IF st_config_achse.b_config_fertig THEN
	(* Fehlermeldungen und Betriebsmeldungen ab dem Startindex in die globalen Meldungsarrays schreiben *)
	garr_stoermeldungen[st_config_achse.i16_meld_startindex + 0] := st_sm.b_achse_nicht_bb;
	garr_stoermeldungen[st_config_achse.i16_meld_startindex + 1] := st_sm.b_achse_nicht_referenziert;
	garr_stoermeldungen[st_config_achse.i16_meld_startindex + 2] := st_sm.b_keine_verfahrfreigabe;
	garr_stoermeldungen[st_config_achse.i16_meld_startindex + 3] := st_sm.b_achse_nicht_auf_startpos;
	garr_stoermeldungen[st_config_achse.i16_meld_startindex + 4] := st_sm.b_ende_skalierungs_nocke;
	garr_stoermeldungen[st_config_achse.i16_meld_startindex + 5] := st_sm.b_ende_camming_nocke;
	garr_stoermeldungen[st_config_achse.i16_meld_startindex + 6] := st_sm.b_skalierung_noch_aktiv;
	garr_stoermeldungen[st_config_achse.i16_meld_startindex + 7] := FALSE;
	garr_stoermeldungen[st_config_achse.i16_meld_startindex + 8] := sm_bandrueckzug;
	garr_stoermeldungen[st_config_achse.i16_meld_startindex + 9] := sm_bandreferenzieren;
	garr_stoermeldungen[st_config_achse.i16_meld_startindex + 10] := sm_fehler_bandvorschub;
	garr_stoermeldungen[st_config_achse.i16_meld_startindex + 11] := sm_fehler_raster;
	garr_stoermeldungen[st_config_achse.i16_meld_startindex + 12] := sm_fehler_bandeinfaedeln;
	garr_stoermeldungen[st_config_achse.i16_meld_startindex + 13] := sm_fahren_auf_gls;
	garr_stoermeldungen[st_config_achse.i16_meld_startindex + 14] := sm_band_rausgezogen;
	garr_stoermeldungen[st_config_achse.i16_meld_startindex + 15] := sm_band_nicht_in_lichtschranke;
	garr_stoermeldungen[st_config_achse.i16_meld_startindex + 16] := st_drive_cmd.meldungen.sm_write_soe_parameter;
	garr_stoermeldungen[st_config_achse.i16_meld_startindex + 17] := st_drive_cmd.meldungen.sm_read_soe_parameter;
	garr_stoermeldungen[st_config_achse.i16_meld_startindex + 18] := st_drive_cmd.meldungen.sm_write_nc_parameter;
	garr_stoermeldungen[st_config_achse.i16_meld_startindex + 19] := st_drive_cmd.meldungen.sm_read_nc_parameter;
	garr_stoermeldungen[st_config_achse.i16_meld_startindex + 20] := st_drive_cmd.meldungen.sm_power_enable;
	garr_stoermeldungen[st_config_achse.i16_meld_startindex + 21] := st_drive_cmd.meldungen.sm_power_disable;
	garr_stoermeldungen[st_config_achse.i16_meld_startindex + 22] := st_drive_cmd.meldungen.sm_reset;
	garr_stoermeldungen[st_config_achse.i16_meld_startindex + 23] := st_drive_cmd.meldungen.sm_home;
	garr_stoermeldungen[st_config_achse.i16_meld_startindex + 24] := st_drive_cmd.meldungen.sm_setposition;
	garr_stoermeldungen[st_config_achse.i16_meld_startindex + 25] := st_drive_cmd.meldungen.sm_jog_vorwaerts;
	garr_stoermeldungen[st_config_achse.i16_meld_startindex + 26] := st_drive_cmd.meldungen.sm_jog_rueckwaerts;
	garr_stoermeldungen[st_config_achse.i16_meld_startindex + 27] := st_drive_cmd.meldungen.sm_move_absolute;
	garr_stoermeldungen[st_config_achse.i16_meld_startindex + 28] := st_drive_cmd.meldungen.sm_move_relative;
	garr_stoermeldungen[st_config_achse.i16_meld_startindex + 29] := st_drive_cmd.meldungen.sm_move_velocity;
	garr_stoermeldungen[st_config_achse.i16_meld_startindex + 30] := st_drive_cmd.meldungen.sm_move_modulo;
	garr_stoermeldungen[st_config_achse.i16_meld_startindex + 31] := st_drive_cmd.meldungen.sm_stop_axis;
	garr_stoermeldungen[st_config_achse.i16_meld_startindex + 32] := st_drive_cmd.meldungen.sm_halt_axis;
	garr_stoermeldungen[st_config_achse.i16_meld_startindex + 33] := st_drive_cmd.meldungen.sm_motion_command_timeout;
	garr_stoermeldungen[st_config_achse.i16_meld_startindex + 34] := st_sm.b_achsfehler;
	garr_stoermeldungen[st_config_achse.i16_meld_startindex + 35] := st_sm.b_devicefehler;
	garr_stoermeldungen[st_config_achse.i16_meld_startindex + 36] := st_drive_cmd.meldungen.sm_limit_positiv_erreicht;
	garr_stoermeldungen[st_config_achse.i16_meld_startindex + 37] := st_drive_cmd.meldungen.sm_limit_negativ_erreicht;
	garr_stoermeldungen[st_config_achse.i16_meld_startindex + 38] := st_drive_cmd.meldungen.sm_ec_coe_sdo_write_ex;
	garr_stoermeldungen[st_config_achse.i16_meld_startindex + 39] := st_drive_cmd.meldungen.sm_ec_coe_sdo_read_ex;
	garr_stoermeldungen[st_config_achse.i16_meld_startindex + 40] := FALSE;
	garr_stoermeldungen[st_config_achse.i16_meld_startindex + 41] := FALSE;
	garr_stoermeldungen[st_config_achse.i16_meld_startindex + 42] := FALSE;
	garr_stoermeldungen[st_config_achse.i16_meld_startindex + 43] := FALSE;
	garr_stoermeldungen[st_config_achse.i16_meld_startindex + 44] := FALSE;
	garr_stoermeldungen[st_config_achse.i16_meld_startindex + 45] := FALSE;
	garr_stoermeldungen[st_config_achse.i16_meld_startindex + 46] := FALSE;
	garr_stoermeldungen[st_config_achse.i16_meld_startindex + 47] := FALSE;
	garr_stoermeldungen[st_config_achse.i16_meld_startindex + 49] := FALSE;
	garr_stoermeldungen[st_config_achse.i16_meld_startindex + 50] := FALSE;
	garr_stoermeldungen[st_config_achse.i16_meld_startindex + 51] := FALSE;
	garr_stoermeldungen[st_config_achse.i16_meld_startindex + 52] := FALSE;
	garr_stoermeldungen[st_config_achse.i16_meld_startindex + 53] := FALSE;
	garr_stoermeldungen[st_config_achse.i16_meld_startindex + 54] := FALSE;
	garr_stoermeldungen[st_config_achse.i16_meld_startindex + 55] := FALSE;
	garr_stoermeldungen[st_config_achse.i16_meld_startindex + 56] := FALSE;
	garr_stoermeldungen[st_config_achse.i16_meld_startindex + 57] := FALSE;
	garr_stoermeldungen[st_config_achse.i16_meld_startindex + 58] := FALSE;
	garr_stoermeldungen[st_config_achse.i16_meld_startindex + 59] := FALSE;
	garr_stoermeldungen[st_config_achse.i16_meld_startindex + 60] := FALSE;
	garr_stoermeldungen[st_config_achse.i16_meld_startindex + 61] := FALSE;
	garr_stoermeldungen[st_config_achse.i16_meld_startindex + 62] := FALSE;
	garr_stoermeldungen[st_config_achse.i16_meld_startindex + 63] := FALSE;
	garr_stoermeldungen[st_config_achse.i16_meld_startindex + 64] := FALSE;
	garr_stoermeldungen[st_config_achse.i16_meld_startindex + 65] := FALSE;
	garr_stoermeldungen[st_config_achse.i16_meld_startindex + 66] := FALSE;
	garr_stoermeldungen[st_config_achse.i16_meld_startindex + 67] := FALSE;
	garr_stoermeldungen[st_config_achse.i16_meld_startindex + 68] := FALSE;
	garr_stoermeldungen[st_config_achse.i16_meld_startindex + 69] := FALSE;
	garr_stoermeldungen[st_config_achse.i16_meld_startindex + 70] := FALSE;
	garr_stoermeldungen[st_config_achse.i16_meld_startindex + 71] := FALSE;
	garr_stoermeldungen[st_config_achse.i16_meld_startindex + 72] := FALSE;
	garr_stoermeldungen[st_config_achse.i16_meld_startindex + 73] := FALSE;
	garr_stoermeldungen[st_config_achse.i16_meld_startindex + 74] := FALSE;
	garr_stoermeldungen[st_config_achse.i16_meld_startindex + 75] := FALSE;
	garr_stoermeldungen[st_config_achse.i16_meld_startindex + 76] := FALSE;
	garr_stoermeldungen[st_config_achse.i16_meld_startindex + 77] := FALSE;
	garr_stoermeldungen[st_config_achse.i16_meld_startindex + 78] := FALSE;
	garr_stoermeldungen[st_config_achse.i16_meld_startindex + 79] := FALSE;
	garr_stoermeldungen[st_config_achse.i16_meld_startindex + 80] := FALSE;
	garr_stoermeldungen[st_config_achse.i16_meld_startindex + 81] := FALSE;
	garr_stoermeldungen[st_config_achse.i16_meld_startindex + 82] := FALSE;
	garr_stoermeldungen[st_config_achse.i16_meld_startindex + 83] := FALSE;
	garr_stoermeldungen[st_config_achse.i16_meld_startindex + 84] := FALSE;
	garr_stoermeldungen[st_config_achse.i16_meld_startindex + 85] := FALSE;
	garr_stoermeldungen[st_config_achse.i16_meld_startindex + 86] := FALSE;
	garr_stoermeldungen[st_config_achse.i16_meld_startindex + 87] := FALSE;
	garr_stoermeldungen[st_config_achse.i16_meld_startindex + 88] := FALSE;
	garr_stoermeldungen[st_config_achse.i16_meld_startindex + 89] := FALSE;
	garr_stoermeldungen[st_config_achse.i16_meld_startindex + 90] := FALSE;
	garr_stoermeldungen[st_config_achse.i16_meld_startindex + 91] := FALSE;
	garr_stoermeldungen[st_config_achse.i16_meld_startindex + 92] := FALSE;
	garr_stoermeldungen[st_config_achse.i16_meld_startindex + 93] := FALSE;
	garr_stoermeldungen[st_config_achse.i16_meld_startindex + 94] := FALSE;
	garr_stoermeldungen[st_config_achse.i16_meld_startindex + 95] := FALSE;
	garr_stoermeldungen[st_config_achse.i16_meld_startindex + 96] := FALSE;
	garr_stoermeldungen[st_config_achse.i16_meld_startindex + 97] := FALSE;
	garr_stoermeldungen[st_config_achse.i16_meld_startindex + 98] := FALSE;
	garr_stoermeldungen[st_config_achse.i16_meld_startindex + 99] := FALSE;
	
	garr_betriebsmeldungen[st_config_achse.i16_meld_startindex + 0] := FALSE;
	garr_betriebsmeldungen[st_config_achse.i16_meld_startindex + 1] := FALSE;
	garr_betriebsmeldungen[st_config_achse.i16_meld_startindex + 2] := FALSE;
	garr_betriebsmeldungen[st_config_achse.i16_meld_startindex + 3] := FALSE;
	garr_betriebsmeldungen[st_config_achse.i16_meld_startindex + 4] := FALSE;
	garr_betriebsmeldungen[st_config_achse.i16_meld_startindex + 5] := FALSE;
	garr_betriebsmeldungen[st_config_achse.i16_meld_startindex + 6] := FALSE;
	garr_betriebsmeldungen[st_config_achse.i16_meld_startindex + 7] := FALSE;
	garr_betriebsmeldungen[st_config_achse.i16_meld_startindex + 8] := FALSE;
	garr_betriebsmeldungen[st_config_achse.i16_meld_startindex + 9] := FALSE;
	garr_betriebsmeldungen[st_config_achse.i16_meld_startindex + 10] := FALSE;
	garr_betriebsmeldungen[st_config_achse.i16_meld_startindex + 11] := FALSE;
	garr_betriebsmeldungen[st_config_achse.i16_meld_startindex + 12] := FALSE;
	garr_betriebsmeldungen[st_config_achse.i16_meld_startindex + 13] := FALSE;
	garr_betriebsmeldungen[st_config_achse.i16_meld_startindex + 14] := FALSE;
	garr_betriebsmeldungen[st_config_achse.i16_meld_startindex + 15] := FALSE;
	garr_betriebsmeldungen[st_config_achse.i16_meld_startindex + 16] := FALSE;
	garr_betriebsmeldungen[st_config_achse.i16_meld_startindex + 17] := FALSE;
	garr_betriebsmeldungen[st_config_achse.i16_meld_startindex + 18] := FALSE;
	garr_betriebsmeldungen[st_config_achse.i16_meld_startindex + 19] := FALSE;
	garr_betriebsmeldungen[st_config_achse.i16_meld_startindex + 20] := FALSE;
	garr_betriebsmeldungen[st_config_achse.i16_meld_startindex + 21] := FALSE;
	garr_betriebsmeldungen[st_config_achse.i16_meld_startindex + 22] := FALSE;
	garr_betriebsmeldungen[st_config_achse.i16_meld_startindex + 23] := FALSE;
	garr_betriebsmeldungen[st_config_achse.i16_meld_startindex + 24] := FALSE;
	garr_betriebsmeldungen[st_config_achse.i16_meld_startindex + 25] := FALSE;
	garr_betriebsmeldungen[st_config_achse.i16_meld_startindex + 26] := FALSE;
	garr_betriebsmeldungen[st_config_achse.i16_meld_startindex + 27] := FALSE;
	garr_betriebsmeldungen[st_config_achse.i16_meld_startindex + 28] := FALSE;
	garr_betriebsmeldungen[st_config_achse.i16_meld_startindex + 29] := FALSE;
	garr_betriebsmeldungen[st_config_achse.i16_meld_startindex + 30] := FALSE;
	garr_betriebsmeldungen[st_config_achse.i16_meld_startindex + 31] := FALSE;
	garr_betriebsmeldungen[st_config_achse.i16_meld_startindex + 32] := FALSE;
	garr_betriebsmeldungen[st_config_achse.i16_meld_startindex + 33] := FALSE;
	garr_betriebsmeldungen[st_config_achse.i16_meld_startindex + 34] := FALSE;
	garr_betriebsmeldungen[st_config_achse.i16_meld_startindex + 35] := FALSE;
	garr_betriebsmeldungen[st_config_achse.i16_meld_startindex + 36] := FALSE;
	garr_betriebsmeldungen[st_config_achse.i16_meld_startindex + 37] := FALSE;
	garr_betriebsmeldungen[st_config_achse.i16_meld_startindex + 38] := FALSE;
	garr_betriebsmeldungen[st_config_achse.i16_meld_startindex + 39] := FALSE;
	garr_betriebsmeldungen[st_config_achse.i16_meld_startindex + 40] := FALSE;
	garr_betriebsmeldungen[st_config_achse.i16_meld_startindex + 41] := FALSE;
	garr_betriebsmeldungen[st_config_achse.i16_meld_startindex + 42] := FALSE;
	garr_betriebsmeldungen[st_config_achse.i16_meld_startindex + 43] := FALSE;
	garr_betriebsmeldungen[st_config_achse.i16_meld_startindex + 44] := FALSE;
	garr_betriebsmeldungen[st_config_achse.i16_meld_startindex + 45] := FALSE;
	garr_betriebsmeldungen[st_config_achse.i16_meld_startindex + 46] := FALSE;
	garr_betriebsmeldungen[st_config_achse.i16_meld_startindex + 47] := FALSE;
	garr_betriebsmeldungen[st_config_achse.i16_meld_startindex + 48] := FALSE;
	garr_betriebsmeldungen[st_config_achse.i16_meld_startindex + 49] := FALSE;
END_IF
END_PROGRAM
ACTION subr_ST_Vorschubkontrolle:
IF gi16_betriebsart <> HAND AND NOT ST_TippTasten.b_einfaedeln_aktiv AND st_ctrl_in.b_freigabe THEN
(* Warte auf Vorschubnocke  und Freigabe von der Virtuellen Masterachse *)
(* Die Freigabe erfolgt nur im normalen Produktionsablauf; nicht bei Bandwechsel, Einfädeln, ... da hier keine Überwachung erfolgen soll. *)

	(* Am Anfang des Bandvorschubs Zähler zurücksetzen *)
	IF  fb_r_trig_nocke_einzug.Q THEN
		i_zaehler_steigende_flanke := 0;
		i_zaehler_fallende_flanke := 0;
	END_IF

	(* Zähler Vorschubkontrolle durch positive Flanke erhöhen *)
	IF fb_r_trig_vorschubkontrolle.Q THEN
		i_zaehler_steigende_flanke := i_zaehler_steigende_flanke + 1;
	END_IF
	(* Zähler Vorschubkontrolle durch negative Flanke erhöhen *)
	IF fb_f_trig_vorschubkontrolle.Q THEN
		i_zaehler_fallende_flanke := i_zaehler_fallende_flanke + 1;
	END_IF

	(* Am Ende des Bandvorschubs die Zähler mit der Vorgabe vergleichen *)
	IF fb_f_trig_nocke_einzug.Q THEN
		IF 	i_zaehler_steigende_flanke <> gst_datensatz.st_bestueckprogramm.i16_b[ST_Virtuelle_Masterachse.i16_bestueckposzaehler] OR
			i_zaehler_fallende_flanke <> gst_datensatz.st_bestueckprogramm.i16_b[ST_Virtuelle_Masterachse.i16_bestueckposzaehler] THEN
			sm_fehler_bandvorschub := TRUE;
			fb_state_entry.i16_next_step := FEHLER;
		END_IF
	END_IF
ELSE
	i_zaehler_steigende_flanke := 0;
	i_zaehler_fallende_flanke := 0;
END_IF
END_ACTION

(* POU Gemeinsamkeiten17xx/Betriebsarten/ST_Betriebsarten, ST *)
PROGRAM ST_Betriebsarten
VAR_INPUT
	st_config					: struct_config;
END_VAR
VAR
	fb_ton_wz				: TON;
	fb_state_entry				: ST_StateEntry;
	i16_betriebsart 			: enum_betriebsarten := KEINE;
	e_ba_automatik			AT %I* : BOOL;
	e_ba_tippen				AT %I* : BOOL;
	e_ba_hand				AT %I* : BOOL;
	e_ba_dummy				AT %I* : BOOL;
	e_ba_pseudo			AT %I* : BOOL;
	a_lampe_ba_automatik	AT %Q* : BOOL;
	a_lampe_ba_tippen		AT %Q* : BOOL;
	a_lampe_ba_hand		AT %Q* : BOOL;
	a_lampe_ba_dummy		AT %Q* : BOOL;
	a_lampe_ba_pseudo		AT %Q* : BOOL;
END_VAR
gi16_betriebsart := i16_betriebsart;

(* Zeiten *)
fb_ton_wz(IN:= , PT:= t#1s, Q=>  , ET=> );

(* ======================================Schrittkette======================================== *)
fb_state_entry(
	i16_next_step:= ,
	i16_pos:= 1,
	s_debugtext:= ,
	E=> ,
	X=> ,
	i16_step=> ,
	i16_last_step=> );

CASE fb_state_entry.i16_step OF
(*=======================================================*)
	0:	(* KEINE *)
		IF fb_state_entry.E THEN
			fb_ton_wz.IN := TRUE;
		END_IF
		IF fb_ton_wz.Q THEN
			i16_betriebsart := KEINE;
		END_IF

		a_lampe_ba_automatik := FALSE;
		a_lampe_ba_tippen := FALSE;
		a_lampe_ba_hand := FALSE;
		a_lampe_ba_dummy := FALSE;
		a_lampe_ba_pseudo := FALSE;

		(* Betriebsartenwechsel *)
		IF e_ba_automatik THEN
			fb_state_entry.i16_next_step := 10;	(* AUTO *)
		ELSIF e_ba_tippen THEN
			fb_state_entry.i16_next_step := 20;	(* TIPPEN *)
		ELSIF e_ba_hand THEN
			fb_state_entry.i16_next_step := 30;	(* HAND *)
		ELSIF e_ba_dummy THEN
			fb_state_entry.i16_next_step := 40;	(* DUMMY *)
		ELSIF e_ba_pseudo THEN
			fb_state_entry.i16_next_step := 50;	(* PSEUDO *)
		END_IF

(*=======================================================*)
	10:	(* AUTO *)
		IF fb_state_entry.E THEN
			i16_betriebsart := AUTO;
			a_lampe_ba_automatik := TRUE;
		END_IF

		(* Betriebsartenwechsel *)
		IF NOT e_ba_automatik THEN
			fb_state_entry.i16_next_step := 0;
		END_IF
	
	(*=======================================================*)
	20:	(* TIPPEN *)
		IF fb_state_entry.E THEN
			i16_betriebsart := TIPPEN;
			a_lampe_ba_tippen := TRUE;
		END_IF

		(* Betriebsartenwechsel *)
		IF NOT e_ba_tippen THEN
			fb_state_entry.i16_next_step := 0;
		END_IF

(*=======================================================*)
	30:	(* HAND *)
		IF fb_state_entry.E THEN
			i16_betriebsart := HAND;
			a_lampe_ba_hand := TRUE;
		END_IF

		(* Betriebsartenwechsel *)
		IF NOT e_ba_hand THEN
			fb_state_entry.i16_next_step := 0;
		END_IF

(*=======================================================*)
	40:	(* DUMMY *)
		IF fb_state_entry.E THEN
			i16_betriebsart := DUMMY;
			a_lampe_ba_dummy := TRUE;
		END_IF

		(* Betriebsartenwechsel *)
		IF NOT e_ba_dummy THEN
			fb_state_entry.i16_next_step := 0;
		END_IF

(*=======================================================*)
	50:	(* PSEUDO *)
		IF fb_state_entry.E THEN
			i16_betriebsart := PSEUDO;
			a_lampe_ba_pseudo := TRUE;
		END_IF

		(* Betriebsartenwechsel *)
		IF NOT e_ba_pseudo THEN
			fb_state_entry.i16_next_step := 0;
		END_IF
END_CASE

fb_state_entry(
	i16_next_step:= ,
	i16_pos:= 2,
	s_debugtext:= ,
	E=> , 
	X=> , 
	i16_step=> ,
	i16_last_step=> );

IF st_config.b_config_fertig THEN
	(* Fehlermeldungen  *)
	garr_stoermeldungen[st_config.i16_meld_startindex + 0] := FALSE;
	garr_stoermeldungen[st_config.i16_meld_startindex + 1] := FALSE;
	garr_stoermeldungen[st_config.i16_meld_startindex + 2] := FALSE;
	garr_stoermeldungen[st_config.i16_meld_startindex + 3] := FALSE;
	garr_stoermeldungen[st_config.i16_meld_startindex + 4] := FALSE;
	garr_stoermeldungen[st_config.i16_meld_startindex + 5] := FALSE;
	garr_stoermeldungen[st_config.i16_meld_startindex + 6] := FALSE;
	garr_stoermeldungen[st_config.i16_meld_startindex + 7] := FALSE;
	garr_stoermeldungen[st_config.i16_meld_startindex + 8] := FALSE;
	garr_stoermeldungen[st_config.i16_meld_startindex + 9] := FALSE;
	garr_stoermeldungen[st_config.i16_meld_startindex + 10] := FALSE;
	garr_stoermeldungen[st_config.i16_meld_startindex + 11] := FALSE;
	garr_stoermeldungen[st_config.i16_meld_startindex + 12] := FALSE;
	garr_stoermeldungen[st_config.i16_meld_startindex + 13] := FALSE;
	garr_stoermeldungen[st_config.i16_meld_startindex + 14] := FALSE;
	garr_stoermeldungen[st_config.i16_meld_startindex + 15] := FALSE;
	garr_stoermeldungen[st_config.i16_meld_startindex + 16] := FALSE;
	garr_stoermeldungen[st_config.i16_meld_startindex + 17] := FALSE;
	garr_stoermeldungen[st_config.i16_meld_startindex + 18] := FALSE;
	garr_stoermeldungen[st_config.i16_meld_startindex + 19] := FALSE;
	
	(* Betriebsmeldungen *)
	garr_betriebsmeldungen[st_config.i16_meld_startindex + 0] := FALSE;
	garr_betriebsmeldungen[st_config.i16_meld_startindex + 1] := FALSE;
	garr_betriebsmeldungen[st_config.i16_meld_startindex + 2] := FALSE;
	garr_betriebsmeldungen[st_config.i16_meld_startindex + 3] := FALSE;
	garr_betriebsmeldungen[st_config.i16_meld_startindex + 4] := FALSE;
	garr_betriebsmeldungen[st_config.i16_meld_startindex + 5] := FALSE;
	garr_betriebsmeldungen[st_config.i16_meld_startindex + 6] := FALSE;
	garr_betriebsmeldungen[st_config.i16_meld_startindex + 7] := FALSE;
	garr_betriebsmeldungen[st_config.i16_meld_startindex + 8] := FALSE;
	garr_betriebsmeldungen[st_config.i16_meld_startindex + 9] := FALSE;
	garr_betriebsmeldungen[st_config.i16_meld_startindex + 10] := FALSE;
	garr_betriebsmeldungen[st_config.i16_meld_startindex + 11] := FALSE;
	garr_betriebsmeldungen[st_config.i16_meld_startindex + 12] := FALSE;
	garr_betriebsmeldungen[st_config.i16_meld_startindex + 13] := FALSE;
	garr_betriebsmeldungen[st_config.i16_meld_startindex + 14] := FALSE;
	garr_betriebsmeldungen[st_config.i16_meld_startindex + 15] := FALSE;
	garr_betriebsmeldungen[st_config.i16_meld_startindex + 16] := FALSE;
	garr_betriebsmeldungen[st_config.i16_meld_startindex + 17] := FALSE;
	garr_betriebsmeldungen[st_config.i16_meld_startindex + 18] := FALSE;
	garr_betriebsmeldungen[st_config.i16_meld_startindex + 19] := FALSE;
END_IF
END_PROGRAM

(* POU Gemeinsamkeiten17xx/Achsen/F_Servobandeinzug_Strecke_zu_Grad, ST *)
FUNCTION F_Servobandeinzug_Strecke_zu_Grad : LREAL
VAR_INPUT
	strecke	: LREAL;
END_VAR
VAR
	Umfang : LREAL;
END_VAR
Umfang :=  gst_datensatz.st_band.i16_igelrad_zaehne * gst_datensatz.st_band.r_raster;
lr_debug :=  (360.0 * strecke ) / Umfang ;
F_Servobandeinzug_Strecke_zu_Grad := lr_debug;
END_FUNCTION

(* POU Gemeinsamkeiten17xx/Achsen/F_Startpos_Servobandeinzug, ST *)
FUNCTION F_Startpos_Servobandeinzug : LREAL
VAR_INPUT
	r_actual_pos : LREAL:= 1.0;
END_VAR
VAR
	i16_gerundet : INT:= 0;
	startpos : INT := 3;
	i16_grad_pro_zahn : INT := 10;
	r_grad_pro_zahn : LREAL := 10.0;
END_VAR
(* Das Igelrad muss zum Einfädeln an einer bestimmten Gradzahl stehen.
Diese ist abhängig von der größe des Igelrads *)

i16_gerundet := LREAL_TO_INT(r_actual_pos/r_grad_pro_zahn);

F_Startpos_Servobandeinzug := INT_TO_LREAL(i16_gerundet * i16_grad_pro_zahn - gst_datensatz.st_band.i16_startpos_einfaedeln);
END_FUNCTION

(* POU Gemeinsamkeiten17xx/TagReader/ST_Konvertiere_gelese_TagData, ST *)
PROGRAM ST_Konvertiere_gelese_TagData
VAR
	i : INT := 0;
END_VAR
IF gst_datensatz.st_md.i16_tag_data_structur_version = 0 THEN
	gst_tag_data.WpcNumber := balluff_tag_reader.fb.s_lese_daten[0];
	gst_tag_data.StateParts[0] := balluff_tag_reader.fb.s_lese_daten[1];
	gst_tag_data.StateParts[1] := balluff_tag_reader.fb.s_lese_daten[2];

	MEMCPY( ADR(gst_tag_data.Articelnumber), ADR(balluff_tag_reader.fb.s_lese_daten[3]), 50);
	gst_tag_data.LastUsedTool := balluff_tag_reader.fb.s_lese_daten[54];
	MEMCPY( ADR(gst_tag_data.UmlNo_VPE), ADR(balluff_tag_reader.fb.s_lese_daten[55]), 4);
	gst_datensatz.st_md.s_aktuelle_artikelnummer := gst_tag_data.Articelnumber;
ELSIF gst_datensatz.st_md.i16_tag_data_structur_version = 1 THEN
	gst_tag_data.WpcNumber := balluff_tag_reader.fb.s_lese_daten[0];
	FOR i:= 0 TO 7 BY 1 DO
		gst_tag_data.StateParts[i] := balluff_tag_reader.fb.s_lese_daten[i + 1];
	END_FOR
	gst_tag_data.AmountPartsOnWpc := balluff_tag_reader.fb.s_lese_daten[10];
	gst_tag_data.LastUsedTool := balluff_tag_reader.fb.s_lese_daten[15];
	MEMCPY( ADR(gst_tag_data.Articelnumber), ADR(balluff_tag_reader.fb.s_lese_daten[20]), 50);
	MEMCPY( ADR(gst_tag_data.UmlNo_VPE), ADR(balluff_tag_reader.fb.s_lese_daten[71]), 4);
	gst_datensatz.st_md.s_aktuelle_artikelnummer := gst_tag_data.Articelnumber;
END_IF

(* Wenn Haken in Visu gesetzt ist dann BESTUECKUNG_MANUAL *)
(* Sonst kommt Info von der WT-XML *)
IF gst_datensatz.st_md.b_bestueckprogramm_manuell THEN
	gst_datensatz.st_md.i16_typ_bestueckmodus := BESTUECKUNG_MANUAL;
ELSE
	gst_datensatz.st_md.i16_typ_bestueckmodus := gst_datensatz.st_wt.i16_typ_bestueckmodus;
END_IF

(* Wenn Hublift links aktiv ist, soll Zelle Last Used Tool auf 0 zurücksetzen *)
(* Damit wird UML simuliert. Diese Funktion ermöglicht Kleinserien mit Hublift links *)
IF gst_datensatz.st_md.b_hublift_links_aktiv THEN
	gst_tag_data.StateParts[0] := PART_NEW;
	gst_tag_data.StateParts[1] := PART_NEW;
	gst_tag_data.LastUsedTool := 0;
END_IF
END_PROGRAM

(* POU Gemeinsamkeiten17xx/TagReader/ST_Markiere_WT_NIO, ST *)
PROGRAM ST_Markiere_WT_NIO
VAR
	i : INT := 0;
END_VAR
IF gst_datensatz.st_md.i16_tag_data_structur_version = 0 THEN
	gst_tag_data.StateParts[0] := PART_NOK;
	gst_tag_data.StateParts[1] := PART_NOK;

	(* Starte Schreib Prozess *)
	balluff_tag_reader.fb.i16_addresse := 1;
	balluff_tag_reader.fb.i16_anzahl_byte := 2;
	balluff_tag_reader.fb.s_schreib_daten[0] := DINT_TO_BYTE(gst_tag_data.StateParts[0]);
	balluff_tag_reader.fb.s_schreib_daten[1] := DINT_TO_BYTE(gst_tag_data.StateParts[1]);
	balluff_tag_reader.st_ctrl.in.b_start_schreiben := TRUE;
ELSIF gst_datensatz.st_md.i16_tag_data_structur_version = 1 THEN
	balluff_tag_reader.fb.i16_addresse := 1;
	balluff_tag_reader.fb.i16_anzahl_byte := 8;
	FOR i:= 0 TO gst_tag_data.AmountPartsOnWpc - 1 BY 1 DO
		gst_tag_data.StateParts[i] := PART_NOK;
	END_FOR
	FOR i:= gst_tag_data.AmountPartsOnWpc TO 7 BY 1 DO
		gst_tag_data.StateParts[i] := PART_NO;
	END_FOR
	FOR i:= 0 TO 7 BY 1 DO
		balluff_tag_reader.fb.s_schreib_daten[i] := DINT_TO_BYTE(gst_tag_data.StateParts[i]);
	END_FOR
	balluff_tag_reader.st_ctrl.in.b_start_schreiben := TRUE;
END_IF
END_PROGRAM

(* POU Gemeinsamkeiten17xx/TagReader/ST_Markiere_WT_IO, ST *)
PROGRAM ST_Markiere_WT_IO
VAR
	i 						:INT := 0;
	b_Rasterfolie_montiert	:BOOL;
END_VAR
(* Auswertung der Bestückung (Pins bzw. Rasterplatte) des ISK *)
CASE gst_datensatz.st_md.i16_typ_zelle OF
	KEINE_ZELLE:
		;

	BESTUECKZELLE_1700:
		(* WT Hat die Maschine auf regulärem Weg wieder verlassen *)
		(* --> Teil ist Ok *)
		IF gst_datensatz.st_md.i16_tag_data_structur_version = 0 THEN
			gst_tag_data.StateParts[0] := PART_OK;
			gst_tag_data.StateParts[1] := PART_OK;	(* Damit die Stuktur nicht umgestellt werden muss, bei 2 ISO auf einem WT *)
		ELSIF gst_datensatz.st_md.i16_tag_data_structur_version = 1 THEN
			FOR i:= 0 TO gst_tag_data.AmountPartsOnWpc - 1 BY 1 DO
				gst_tag_data.StateParts[i] := PART_OK;
			END_FOR
			FOR i:= gst_tag_data.AmountPartsOnWpc TO 7 BY 1 DO
				gst_tag_data.StateParts[i] := PART_NO;
			END_FOR
		END_IF

	BESTUECKZELLE_1720:
		(* WT Hat die Maschine auf regulärem Weg wieder verlassen *)
		(* --> Teil ist Ok *)
		IF gst_datensatz.st_md.i16_tag_data_structur_version = 0 THEN
			gst_tag_data.StateParts[0] := PART_OK;
			gst_tag_data.StateParts[1] := PART_OK;
		ELSIF gst_datensatz.st_md.i16_tag_data_structur_version = 1 THEN
			FOR i:= 0 TO gst_tag_data.AmountPartsOnWpc - 1 BY 1 DO
				gst_tag_data.StateParts[i] := PART_OK;
			END_FOR
			FOR i:= gst_tag_data.AmountPartsOnWpc TO 7 BY 1 DO
				gst_tag_data.StateParts[i] := PART_NO;
			END_FOR
		END_IF

	RASTERFOLIE:
			b_Rasterfolie_montiert:=	TRUE;
			FOR i := 0 TO DINT_TO_INT(gst_datensatz.st_bestueckprogramm.i32_anzahl) - 1 BY 1 DO
				IF	NOT ST_Rasterfolienmontage.arr_rafo_schieberegister[i]THEN
					b_Rasterfolie_montiert:=	FALSE;
				END_IF
			END_FOR

		IF gst_datensatz.st_md.i16_tag_data_structur_version = 0 THEN
			IF b_Rasterfolie_montiert THEN
				gst_tag_data.StateParts[0] := PART_OK;
				gst_tag_data.StateParts[1] := PART_OK;	(* Damit die Stuktur nicht umgestellt werden muss, bei 2 ISO auf einem WT *)
			ELSE
				gst_tag_data.StateParts[0] := PART_NOK;
				gst_tag_data.StateParts[1] := PART_NOK;
			END_IF
		ELSIF gst_datensatz.st_md.i16_tag_data_structur_version = 1 THEN
			IF b_Rasterfolie_montiert THEN
				FOR i:= 0 TO gst_tag_data.AmountPartsOnWpc - 1 BY 1 DO
					gst_tag_data.StateParts[i] := PART_OK;
				END_FOR
				FOR i:= gst_tag_data.AmountPartsOnWpc TO 7 BY 1 DO
					gst_tag_data.StateParts[i] := PART_NO;
				END_FOR
			ELSE
				FOR i:= 0 TO gst_tag_data.AmountPartsOnWpc - 1 BY 1 DO
					gst_tag_data.StateParts[i] := PART_NOK;
				END_FOR
				FOR i:= gst_tag_data.AmountPartsOnWpc TO 7 BY 1 DO
					gst_tag_data.StateParts[i] := PART_NO;
				END_FOR
			END_IF
		END_IF
END_CASE
(* Starte Schreib Prozess *)
IF gst_datensatz.st_md.i16_tag_data_structur_version = 0 THEN
	balluff_tag_reader.fb.i16_addresse := 1;
	balluff_tag_reader.fb.i16_anzahl_byte := 2;
	balluff_tag_reader.fb.s_schreib_daten[0] := DINT_TO_BYTE(gst_tag_data.StateParts[0]);
	balluff_tag_reader.fb.s_schreib_daten[1] := DINT_TO_BYTE(gst_tag_data.StateParts[1]);
	balluff_tag_reader.st_ctrl.in.b_start_schreiben := TRUE;
ELSIF gst_datensatz.st_md.i16_tag_data_structur_version = 1THEN
	balluff_tag_reader.fb.i16_addresse := 1;
	balluff_tag_reader.fb.i16_anzahl_byte := 8;
	FOR i:= 0 TO 7 BY 1 DO
		balluff_tag_reader.fb.s_schreib_daten[i] := DINT_TO_BYTE(gst_tag_data.StateParts[i]);
	END_FOR
	balluff_tag_reader.st_ctrl.in.b_start_schreiben := TRUE;
END_IF
END_PROGRAM

(* POU Gemeinsamkeiten17xx/TagReader/ST_Schreibe_LastUsedTool, ST *)
PROGRAM ST_Schreibe_LastUsedTool
VAR
END_VAR
(* Starte Schreib Prozess *)
IF gst_datensatz.st_md.i16_tag_data_structur_version = 0 THEN
	balluff_tag_reader.fb.i16_addresse := 54;
	balluff_tag_reader.fb.i16_anzahl_byte := 1;
	balluff_tag_reader.fb.s_schreib_daten[0] := gst_tag_data.LastUsedTool;
	balluff_tag_reader.st_ctrl.in.b_start_schreiben := TRUE;
ELSIF gst_datensatz.st_md.i16_tag_data_structur_version = 1 THEN
	balluff_tag_reader.fb.i16_addresse := 15;
	balluff_tag_reader.fb.i16_anzahl_byte := 1;
	balluff_tag_reader.fb.s_schreib_daten[0] := gst_tag_data.LastUsedTool;
	balluff_tag_reader.st_ctrl.in.b_start_schreiben := TRUE;
END_IF
END_PROGRAM

(* POU Gemeinsamkeiten17xx/Achsen/ST_Bestueckachse, ST *)
PROGRAM ST_Bestueckachse
VAR_INPUT
	st_config_achse						: struct_ecd_config;
	st_ctrl_in								: struct_ctrl_in;
	e_steuerung_ein						: BOOL;
	e_ba_mit_bedingungen				: BOOL;
	e_tuere_vorne_offen					: BOOL;
	e_tuere_hinten_offen					: BOOL;
END_VAR
VAR_IN_OUT
	st_visu								: struct_ecd_visu;
END_VAR
VAR_OUTPUT
	st_ctrl_out							: struct_ctrl_out;
END_VAR
VAR
	st_sm						 		: struct_ecd_meldungen;
	st_drive_cmd							: struct_ecd_cmd;
	fb_ton_wz							: TON;
	fb_ton_quitt							: TON;
	fb_ton_wz_disable						: TON;
	fb_r_trig_tippen						: R_TRIG;
	fb_f_trig_tippen						: F_TRIG;
	fb_r_trig_taste_plus					: R_TRIG;
	fb_r_trig_taste_minus					: R_TRIG;
	fb_r_trig_start							: R_TRIG;
	fb_r_trig_hand_dialog					: R_TRIG;
	fb_r_trig_nullpunkt_setzen				: R_TRIG;
	fb_axis								: ST_AxisJobCtrl_Motion;
	fb_state_entry							: ST_StateEntry;
	fb_ton_uez							: TON;
	i, j									: INT := 0;
	lr_pos_ohneverschiebung			: LREAL;
	st_geschwindigkeiten					: struct_ecd_geschwindigkeiten;
	b_hand_dialog_aktiv					: BOOL := FALSE;
	b_nullnockenmerker					: BOOL := FALSE;

	sm_fehler_initialposition_achse			: BOOL := FALSE;
	sm_keine_nocken_definiert				: BOOL := FALSE;
	sm_fehler_ot_ut						: BOOL := FALSE;

	e_referenz_sensor						AT %I* : BOOL;
	i16_torque							AT %I* : INT;

	fb_ot_ut_ueberwachung				: ST_OT_UT_Ueberwachung;

	lr_decceleration_nothalt				: LREAL;
	lr_decceleration_normal				: LREAL;
END_VAR
(* Zeiten *)
fb_ton_wz(IN:= ,PT:= , Q=>  , ET=> );
fb_ton_uez(IN:= ,	PT:= , Q=>  , ET=> );
fb_ton_quitt(IN:= , PT:= t#100ms, Q=> , ET=> );
fb_ton_wz_disable(IN:= , PT:= t#500ms, Q=> , ET=> );

(* Flanken *)
fb_r_trig_taste_plus(CLK:= ST_Euchner_Handbedienpult.b_Taste_Plus, Q=> );
fb_r_trig_taste_minus(CLK:= ST_Euchner_Handbedienpult.b_Taste_Minus, Q=> );
fb_r_trig_start(CLK:= st_ctrl_in.b_start, Q=> );
fb_r_trig_hand_dialog(CLK:= b_hand_dialog_aktiv, Q=> );
fb_r_trig_nullpunkt_setzen(CLK:= axis_bestueckachse.st_visu.b_nullpunkt_setzen, Q=> );

(* Achse steuern *)
(* Bestueckachse *)
fb_axis(
	e_referenznocken:= ,
	b_refsensor_vorhanden:= st_config_achse.b_refsensor_vorhanden,
	b_limitsensor_positiv_vorhanden:= st_config_achse.b_limitsensor_positiv_vorhanden,
	b_limitsensor_negativ_vorhanden:= st_config_achse.b_limitsensor_negativ_vorhanden,
	i16_achstyp := st_config_achse.i16_achstyp,
	st_position:= ,
	lr_override_vorgabe:= ST_TippTasten.lr_override,
	mc_richtung_modulo:= ,
	mc_richtung_velocity:= ,
	mc_referenzmodus:= ,
	mc_buffermode_axis:= ,
	ui16_soeparam_write_value:= ,
	w_idn:= ,
	i16_nc_parameter_nummer:= ,
	r_wert_nc_write_parameter:= ,
	st_vorgabe_geschwindigkeiten:= st_geschwindigkeiten,
	lr_soll_geschwindigkeit:=,
	b_bedingung_sls:= NOT e_tuere_vorne_offen OR NOT e_tuere_hinten_offen,
	st_ads_info := ,
	st_eccoe_sdo := ,
	st_masterachse:= bestueckachse,
	st_visu_axis:= st_visu,
	st_ecd_cmd:= st_drive_cmd,
	ui16_soeparam_read_value=> ,
	r_wert_nc_read_parameter=> );

IF gi16_betriebsart <> AUTO THEN
	(* Bausteinaufruf für Kontrolle der korrekten Abfolge von OT zu UT. Nicht für Automatikbetrieb geeignet, da Aufruf in der normalen Task! *)
	fb_ot_ut_ueberwachung(
		lr_achsposition:= bestueckachse.NcToPlc.ModuloActPos,
		b_error=> sm_fehler_ot_ut);
ELSE
	sm_fehler_ot_ut := FALSE;
END_IF

IF gi16_betriebsart = HAND THEN
	(* Achse mit dem Euchner Handbediengerät vorwärts und rückwärts Bewegen*)
	IF fb_r_trig_hand_dialog.Q THEN
		fb_state_entry.i16_next_step := HANDRAD;
	END_IF

	(* Button in der Oberfläche zum setzen des Nullpunktes *)
	IF fb_r_trig_nullpunkt_setzen.Q THEN
		fb_state_entry.i16_next_step :=	NULLPUNKT_SETZEN;
	END_IF
END_IF


(* =======================================Toplevel========================================== *)
(* Starte Inbetriebnahme-Sequenz *)
IF st_ctrl_in.b_gehe_step_ibn THEN
	fb_state_entry.i16_next_step := INBETRIEBNAHME;
END_IF

(* =====Achse wird disabled===== *)
IF (NOT e_steuerung_ein OR NOT e_ba_mit_bedingungen) AND bestueckachse.Status.Operational THEN
	st_drive_cmd.enu_cmd := POWER_DISABLE;
END_IF

IF fb_state_entry.i16_next_step > INIT AND fb_state_entry.i16_next_step < FEHLER THEN
	(* =====Fehler vom Achskontroller===== *)
	IF st_drive_cmd.b_job_fehler THEN
		fb_state_entry.i16_next_step := FEHLER;
	END_IF

	IF fb_state_entry.i16_next_step > 45 THEN
		(* Devicefehler *)
		IF bestueckachse.Status.Error THEN
			st_sm.b_achsfehler := TRUE;
			fb_state_entry.i16_next_step := FEHLER;
		ELSIF bestueckachse.Status.DriveDeviceError THEN
			st_sm.b_devicefehler := TRUE;
			fb_state_entry.i16_next_step := FEHLER;
		END_IF
	END_IF

	IF fb_state_entry.i16_next_step < STOP THEN
		(* =====Achse wird gestoppt===== *)
		IF st_ctrl_in.b_stop THEN
			fb_state_entry.i16_next_step := STOP;
		ELSIF fb_state_entry.i16_next_step < HALT THEN
			(* =====Achse wird angehalten===== *)
			IF st_ctrl_in.b_halt THEN
				fb_state_entry.i16_next_step := HALT;
			END_IF
		END_IF
	END_IF
END_IF

(* ======================================Schrittkette======================================== *)
fb_state_entry(
	i16_next_step:= ,
	i16_pos:= 1,
	s_debugtext:= ,
	E=> ,
	X=> ,
	i16_step=> ,
	i16_last_step=> );

CASE fb_state_entry.i16_step OF
(*=======================================================*)
	INIT_OBJ:
		IF st_config_achse.b_config_fertig THEN
			fb_state_entry.i16_next_step := 1;
		END_IF

(*=======================================================*)
	1:	(* Warte bis NetID´s der Slaves ausgelesen sind *)
		IF fb_state_entry.E THEN
			;
		END_IF

		(*-----------------------Weiterschaltbedingungen----------------------------*)
		IF ST_EthercatDiag.st_ctrl_out.b_fertig THEN
			fb_state_entry.i16_next_step := 3;
		END_IF

(*=======================================================*)
	3:	(* Spezifische NC-Achsparameter auslesen *)
		IF fb_state_entry.E THEN
			FOR i := 0  TO (SIZEOF (nockenschaltwerk_bestueckachse.fb.arr_spur) / SIZEOF (nockenschaltwerk_bestueckachse.fb.arr_spur[0])) - 1 BY 1DO
				gst_datensatz.st_wkz.nockenschaltwerk_bestueckachse.arr_nocken[i].b_camvalid := TRUE;
			END_FOR

			fb_axis.i16_nc_parameter_nummer := MaxVelocitySystem;
			st_drive_cmd.enu_cmd := READ_NC_PARAMETER;
		END_IF

		(*-----------------------Weiterschaltbedingungen----------------------------*)
		IF st_drive_cmd.enu_cmd = NO_COMMAND THEN
			st_geschwindigkeiten.lr_maximalgeschwindigkeit := fb_axis.r_wert_nc_read_parameter(* °/s *) * 60 / 360;
			st_geschwindigkeiten.lr_auto_max := st_geschwindigkeiten.lr_maximalgeschwindigkeit;
			st_geschwindigkeiten.lr_auto_min := 50;
			st_geschwindigkeiten.lr_jog := 100;
			fb_state_entry.i16_next_step := 4;
		END_IF

(*=======================================================*)
	4:	(* Spezifische NC-Achsparameter auslesen *)
		IF fb_state_entry.E THEN
			fb_axis.i16_nc_parameter_nummer := MaxAccelerationSystem;
			st_drive_cmd.enu_cmd := READ_NC_PARAMETER;
		END_IF

		(*-----------------------Weiterschaltbedingungen----------------------------*)
		IF st_drive_cmd.enu_cmd = NO_COMMAND THEN
			st_geschwindigkeiten.lr_beschleunigung := fb_axis.r_wert_nc_read_parameter;
			fb_state_entry.i16_next_step := 5;
		END_IF

(*=======================================================*)
	5:	(* Spezifische NC-Achsparameter auslesen *)
		IF fb_state_entry.E THEN
			fb_axis.i16_nc_parameter_nummer := MaxDecelerationSystem;
			st_drive_cmd.enu_cmd := READ_NC_PARAMETER;
		END_IF

		(*-----------------------Weiterschaltbedingungen----------------------------*)
		IF st_drive_cmd.enu_cmd = NO_COMMAND THEN
			st_geschwindigkeiten.lr_verzoegerung := fb_axis.r_wert_nc_read_parameter;
			lr_decceleration_normal := st_geschwindigkeiten.lr_verzoegerung;
			lr_decceleration_nothalt := 200000.0;
			fb_state_entry.i16_next_step := 6;
		END_IF

(*=======================================================*)
	6:	(* Spezifische NC-Achsparameter auslesen *)
		IF fb_state_entry.E THEN
			fb_axis.i16_nc_parameter_nummer := MaxJerk;
			st_drive_cmd.enu_cmd := READ_NC_PARAMETER;
		END_IF

		(*-----------------------Weiterschaltbedingungen----------------------------*)
		IF st_drive_cmd.enu_cmd = NO_COMMAND THEN
			st_geschwindigkeiten.lr_ruck := fb_axis.r_wert_nc_read_parameter;
			fb_state_entry.i16_next_step := 7;
		END_IF

(*=======================================================*)
	7:	(* Konfigurationen der Achse *)
		IF fb_state_entry.E THEN
			fb_axis.st_eccoe_sdo.s_ec_slave_net_id := ST_EthercatDiag.s_ec_slave_net_id[2];
			fb_axis.st_eccoe_sdo.ui16_slave_addr := st_config_achse.ui16_ethercat_adr;
		END_IF

		(*-----------------------Weiterschaltbedingungen----------------------------*)
		fb_state_entry.i16_next_step := FEHLER; (*in Fehler gehen damit die Achsen resetet werden. Sonst steigen die Achsen bei einem TC Restart aus*)

(*=======================================================*)
	INIT:
		IF fb_state_entry.E THEN
			fb_ton_wz.IN := FALSE;
			fb_ton_uez.IN	:= FALSE;
			fb_ton_quitt.IN := FALSE;
			fb_ton_wz_disable.IN := FALSE;
			st_ctrl_out.b_fehler := FALSE;
			st_ctrl_out.b_fertig := FALSE;
			st_ctrl_out.b_bereit := FALSE;
			st_ctrl_out.b_prebereit := FALSE;

 			fb_axis.lr_soll_geschwindigkeit := gst_datensatz.st_wkz.r_auto;

			st_geschwindigkeiten.lr_verzoegerung := lr_decceleration_normal;

			(* Reset Stoermeldungen *)
			st_sm.b_achse_nicht_auf_startpos := FALSE;
			st_sm.b_achsfehler := FALSE;
			st_sm.b_devicefehler := FALSE;
			st_sm.b_keine_verfahrfreigabe := FALSE;
			st_sm.b_ende_skalierungs_nocke := FALSE;
			st_sm.b_ende_camming_nocke := FALSE;
			st_sm.b_skalierung_noch_aktiv := FALSE;

			sm_fehler_initialposition_achse := FALSE;
			sm_keine_nocken_definiert := FALSE;

		END_IF

		(*-----------------------Weiterschaltbedingungen----------------------------*)
		IF st_ctrl_in.b_preinit THEN
			fb_axis.lr_soll_geschwindigkeit := gst_datensatz.st_wkz.r_auto;
			fb_state_entry.i16_next_step := 15;
		END_IF

(*=======================================================*)
	15:	(* Reglerfreigabe wegnehmen *)
		IF fb_state_entry.E THEN
			st_drive_cmd.enu_cmd := POWER_DISABLE;
		END_IF

		(*-----------------------Weiterschaltbedingungen----------------------------*)
		IF st_drive_cmd.enu_cmd = NO_COMMAND THEN
			fb_state_entry.i16_next_step := 20;
		END_IF

(*=======================================================*)
	20:	(* Überprüfe Nullpunktverschiebung des Absolutwertgebers auf Korrektheit *)
		IF fb_state_entry.E THEN
			fb_axis.i16_nc_parameter_nummer := AxisEncoderOffset;	(* vom Datentyp MC_AxisParameter *)
			st_drive_cmd.enu_cmd := READ_NC_PARAMETER;
		END_IF

		(*-----------------------Weiterschaltbedingungen----------------------------*)
		IF st_drive_cmd.enu_cmd = NO_COMMAND THEN
			IF fb_axis.r_wert_nc_read_parameter = gst_datensatz.st_md.st_md_bestueckachse.lr_nullpunktverschiebung THEN
				fb_state_entry.i16_next_step := 45;	(* Reglerfreigabe setzen *)
			ELSE
				fb_state_entry.i16_next_step := 30;	(* Nullpunktverschiebung schreiben *)
			END_IF
		END_IF
(*
(*=======================================================*)
	25:	(* Überprüfung der Achsposition mit Referenzsensor *)

		(*-----------------------Weiterschaltbedingungen----------------------------*)
		IF e_referenz_sensor THEN
			fb_state_entry.i16_next_step := 30;	(* Achse steht im korrekten Winkelbereich *)
		ELSE
			sm_fehler_initialposition_achse := TRUE;
			fb_state_entry.i16_next_step := FEHLER;	(* Achsposition ist um Vielfache von 72° verschoben *)
		END_IF
*)
(*=======================================================*)
	30:	(* Nullpunktverschiebung hat sich geändert, deshalb erst Null reinschreiben, um keinen Additionsfehler zu machen, *)
		(* weil der Wert der Verschiebung beim Neustart komplett auf die Achse geschrieben wird *)
		IF fb_state_entry.E THEN
			fb_axis.i16_nc_parameter_nummer := AxisEncoderOffset;
			fb_axis.r_wert_nc_write_parameter := 0.0;
			st_drive_cmd.enu_cmd := WRITE_NC_PARAMETER;
		END_IF

		(*-----------------------Weiterschaltbedingungen----------------------------*)
		IF st_drive_cmd.enu_cmd = NO_COMMAND THEN
			fb_state_entry.i16_next_step := 40;
		END_IF

(*=======================================================*)
	40:	(* Aktuelle Nullpunktverschiebung des Absolutwertgebers an die Achse senden *)
		IF fb_state_entry.E THEN
			fb_axis.i16_nc_parameter_nummer := AxisEncoderOffset;
			fb_axis.r_wert_nc_write_parameter := gst_datensatz.st_md.st_md_bestueckachse.lr_nullpunktverschiebung;
			st_drive_cmd.enu_cmd := WRITE_NC_PARAMETER;
		END_IF

		(*-----------------------Weiterschaltbedingungen----------------------------*)
		IF st_drive_cmd.enu_cmd = NO_COMMAND THEN
			fb_state_entry.i16_next_step := 45;
		END_IF

(*=======================================================*)
	45:	(* Reglerfreigabe setzen , Reset wird bei Bedarf automatisch ausgeführt*)
		IF fb_state_entry.E THEN
			st_drive_cmd.enu_cmd := POWER_ENABLE;
		END_IF

		(*-----------------------Weiterschaltbedingungen----------------------------*)
		IF st_drive_cmd.enu_cmd = NO_COMMAND THEN
			fb_state_entry.i16_next_step := 50;
		END_IF

(*=======================================================*)
	50:
		IF fb_state_entry.E THEN
			st_ctrl_out.b_prebereit := TRUE;
		END_IF

		(*-----------------------Weiterschaltbedingungen----------------------------*)
		IF st_ctrl_in.b_init THEN
			fb_state_entry.i16_next_step := 60;
		END_IF

(*=======================================================*)
	60:	(* Überprüfe, ob überhaupt Nocken angelegt sind *)
		IF fb_state_entry.E THEN
			b_nullnockenmerker := TRUE;
			FOR i := 0  TO 5 BY 1DO
				b_nullnockenmerker :=	b_nullnockenmerker AND
								 	gst_datensatz.st_wkz.nockenschaltwerk_bestueckachse.arr_nocken[i].r_cam_begin = 0 AND
									gst_datensatz.st_wkz.nockenschaltwerk_bestueckachse.arr_nocken[i].r_cam_end = 0;
			END_FOR
		END_IF

		(*-----------------------Weiterschaltbedingungen----------------------------*)
		IF b_nullnockenmerker	THEN
			sm_keine_nocken_definiert := TRUE;
			 fb_state_entry.i16_next_step := FEHLER;
		ELSE
			fb_state_entry.i16_next_step := 70;
		END_IF

(*=======================================================*)
	70: (* Alle Nocken einschalten *)
		IF fb_state_entry.E THEN
			FOR i := 0  TO (SIZEOF (nockenschaltwerk_bestueckachse.fb.arr_spur) / SIZEOF (nockenschaltwerk_bestueckachse.fb.arr_spur[0])) - 1 BY 1DO
				gst_datensatz.st_wkz.nockenschaltwerk_bestueckachse.arr_nocken[i].b_camvalid := TRUE;
				gst_datensatz.st_wkz.nockenschaltwerk_bestueckachse.arr_nocken[i].b_eff_direction_neg := TRUE;
				gst_datensatz.st_wkz.nockenschaltwerk_bestueckachse.arr_nocken[i].b_eff_direction_pos := TRUE;
				gst_datensatz.st_wkz.nockenschaltwerk_bestueckachse.arr_nocken[i].i16_track_no := i;
			END_FOR
			(* Nachbearbeitung von bestimmten Nocken *)
			gst_datensatz.st_wkz.nockenschaltwerk_bestueckachse.arr_nocken[NO_OT].b_eff_direction_neg := FALSE;

			(* Zylinder für Bandeinzug mit Vorsteuerzeit belegen *)
			(* 1700 *)
			CASE gst_datensatz.st_wkz.i16_typ_bandeinzug OF
				KEIN_EINZUG:
					;

				STANDARD_2FACH_V2:
					gst_datensatz.st_wkz.nockenschaltwerk_bestueckachse.arr_nocken[NO_BW_BANDFAENGER_LI_BAEZV2_EINFAHREN].t_vorsteuerzeit := t#16ms;
					gst_datensatz.st_wkz.nockenschaltwerk_bestueckachse.arr_nocken[NO_BW_BANDFAENGER_LI_BAEZV2_AUSFAHREN].t_vorsteuerzeit := t#16ms;
					gst_datensatz.st_wkz.nockenschaltwerk_bestueckachse.arr_nocken[NO_BW_BANDKLEMMEN_LI_BAEZV2_EINFAHREN].t_vorsteuerzeit := t#16ms;
					gst_datensatz.st_wkz.nockenschaltwerk_bestueckachse.arr_nocken[NO_BW_BANDKLEMMEN_LI_BAEZV2_AUSFAHREN].t_vorsteuerzeit := t#16ms;
					gst_datensatz.st_wkz.nockenschaltwerk_bestueckachse.arr_nocken[NO_BW_BANDFAENGER_RE_BAEZV2_EINFAHREN].t_vorsteuerzeit := t#16ms;
					gst_datensatz.st_wkz.nockenschaltwerk_bestueckachse.arr_nocken[NO_BW_BANDFAENGER_RE_BAEZV2_AUSFAHREN].t_vorsteuerzeit := t#16ms;
					gst_datensatz.st_wkz.nockenschaltwerk_bestueckachse.arr_nocken[NO_BW_BANDKLEMMEN_RE_BAEZV2_EINFAHREN].t_vorsteuerzeit := t#16ms;
					gst_datensatz.st_wkz.nockenschaltwerk_bestueckachse.arr_nocken[NO_BW_BANDKLEMMEN_RE_BAEZV2_AUSFAHREN].t_vorsteuerzeit := t#16ms;

				BANDWECHSLER_V2:
					(* Bandwechsler V2 ohne Sensoren und anderen Zylindern *)
					gst_datensatz.st_wkz.nockenschaltwerk_bestueckachse.arr_nocken[NO_BW_BANDFAENGER_BAWEV2_EINFAHREN].t_vorsteuerzeit := t#16ms;
					gst_datensatz.st_wkz.nockenschaltwerk_bestueckachse.arr_nocken[NO_BW_BANDFAENGER_BAWEV2_AUSFAHREN].t_vorsteuerzeit := t#16ms;
					gst_datensatz.st_wkz.nockenschaltwerk_bestueckachse.arr_nocken[NO_BW_BANDKLEMMEN_BAWEV2_EINFAHREN].t_vorsteuerzeit := t#16ms;
					gst_datensatz.st_wkz.nockenschaltwerk_bestueckachse.arr_nocken[NO_BW_BANDKLEMMEN_BAWEV2_AUSFAHREN].t_vorsteuerzeit := t#16ms;

				SERVO:
					;
(*					gst_datensatz.st_wkz.nockenschaltwerk_bestueckachse.arr_nocken[NO_SERVOBANDEINZUG_LUEFTEN].r_cam_begin := 135;
					gst_datensatz.st_wkz.nockenschaltwerk_bestueckachse.arr_nocken[NO_SERVOBANDEINZUG_LUEFTEN].r_cam_end := 178;
					gst_datensatz.st_wkz.nockenschaltwerk_bestueckachse.arr_nocken[NO_SERVOBANDEINZUG_GLS].r_cam_begin := 50;
					gst_datensatz.st_wkz.nockenschaltwerk_bestueckachse.arr_nocken[NO_SERVOBANDEINZUG_GLS].r_cam_end := 100;*)
			END_CASE;

			(*-----------------------Weiterschaltbedingungen----------------------------*)
			fb_state_entry.i16_next_step := 80;
		END_IF

(*=======================================================*)
	80:  (* Auf Startposition fahren *)
		CASE gst_datensatz.st_md.i16_typ_zelle OF
			KEINE_ZELLE:
				;

			BESTUECKZELLE_1700, RASTERFOLIE:
				IF fb_state_entry.E THEN
					st_drive_cmd.enu_cmd := MOVE_MODULO;
					fb_axis.mc_richtung_modulo := MC_Shortest_Way ;
					fb_axis.st_position.r_soll := gst_datensatz.st_md.st_md_bestueckachse.lr_startposition;
				END_IF

			BESTUECKZELLE_1720:
				IF fb_state_entry.E THEN
					IF bestueckachse.NcToPlc.ModuloActPos > 0 AND bestueckachse.NcToPlc.ModuloActPos < 90 THEN
						fb_axis.mc_richtung_modulo := MC_Shortest_Way ;
					ELSE
						fb_axis.mc_richtung_modulo := MC_Positive_Direction;
					END_IF
					st_drive_cmd.enu_cmd := MOVE_MODULO;
					fb_axis.st_position.r_soll := gst_datensatz.st_md.st_md_bestueckachse.lr_startposition;
				END_IF
		END_CASE

		(*-----------------------Weiterschaltbedingungen----------------------------*)
		IF st_drive_cmd.enu_cmd = NO_COMMAND THEN
			fb_state_entry.i16_next_step := 90;
		END_IF

(*=======================================================*)
	90:	(* Finale Überprüfung der Achsposition auf Bereich OT oder UT *)

		(*-----------------------Weiterschaltbedingungen----------------------------*)
		IF e_referenz_sensor AND
			bestueckachse.NcToPlc.ModuloActPos >= 0 AND
			bestueckachse.NcToPlc.ModuloActPos < 71.99 THEN
			fb_state_entry.i16_next_step := BEREIT;	(* Achse steht im korrekten Winkelbereich *)
		ELSE
			sm_fehler_initialposition_achse := TRUE;
			fb_state_entry.i16_next_step := FEHLER;	(* Achsposition ist um Vielfache von 72° verschoben *)
		END_IF

(*=======================================================*)
	BEREIT:
		IF fb_state_entry.E THEN
			st_ctrl_out.b_bereit := TRUE;
			st_ctrl_out.b_fertig := TRUE;
		END_IF

(*=======================================================*)
	FEHLER:
		IF fb_state_entry.E THEN
			st_ctrl_out.b_fehler := TRUE;
			fb_ton_quitt.IN := FALSE;
		END_IF

		(*-----------------------Weiterschaltbedingungen----------------------------*)
		IF st_ctrl_in.b_quitt AND NOT fb_state_entry.E THEN
			st_ctrl_out.b_fehler := FALSE;
			st_drive_cmd.enu_cmd := RESET;
			fb_ton_quitt.IN := TRUE;
		END_IF

		IF st_ctrl_in.b_stop AND NOT bestueckachse.Status.HasBeenStopped THEN
			st_drive_cmd.enu_cmd := STOP_AXIS;
		END_IF

		IF st_ctrl_in.b_halt AND bestueckachse.Status.Moving THEN
			st_drive_cmd.enu_cmd := HALT_AXIS;
			st_geschwindigkeiten.lr_verzoegerung := lr_decceleration_nothalt;
		END_IF

		IF fb_ton_quitt.Q THEN
			fb_ton_quitt.IN := FALSE;
			fb_state_entry.i16_next_step := INIT;
		END_IF

(*=======================================================*)
	STOP:
		IF fb_state_entry.E THEN
			IF bestueckachse.NcToPlc.CoupleState = 0 THEN
				st_drive_cmd.enu_cmd := STOP_AXIS;
			END_IF
		END_IF

		(*-----------------------Weiterschaltbedingungen----------------------------*)
		IF st_drive_cmd.enu_cmd = NO_COMMAND AND bestueckachse.Status.NotMoving THEN
			fb_state_entry.i16_next_step := STILLSTAND;
		END_IF

(*=======================================================*)
	STILLSTAND:
		IF fb_state_entry.E THEN
			st_drive_cmd.enu_cmd := POWER_DISABLE;
			fb_ton_quitt.IN := FALSE;
		END_IF

		(*-----------------------Weiterschaltbedingungen----------------------------*)
		IF st_ctrl_in.b_quitt AND NOT fb_state_entry.E THEN
			fb_ton_quitt.IN := TRUE;
		END_IF

		IF fb_ton_quitt.Q THEN
			fb_ton_quitt.IN := FALSE;
			fb_state_entry.i16_next_step := INIT;
		END_IF

(*=======================================================*)
	HALT:
		IF fb_state_entry.E THEN
			IF bestueckachse.NcToPlc.CoupleState = 0 THEN
				st_drive_cmd.enu_cmd := HALT_AXIS;
				st_geschwindigkeiten.lr_verzoegerung := lr_decceleration_nothalt;
			END_IF
			fb_ton_quitt.IN := FALSE;
		END_IF

		(*-----------------------Weiterschaltbedingungen----------------------------*)
		IF st_ctrl_in.b_quitt AND NOT fb_state_entry.E THEN
			fb_ton_quitt.IN := TRUE;
		END_IF

		IF fb_ton_quitt.Q THEN
			fb_ton_quitt.IN := FALSE;
			fb_state_entry.i16_next_step := INIT;
		END_IF

(*=======================================================*)
	HANDRAD:	(* Überprüfe Nullpunktverschiebung des Absolutwertgebers auf Korrektheit *)
		IF fb_state_entry.E THEN
			st_ctrl_out.b_fehler := TRUE;
			fb_axis.i16_nc_parameter_nummer := AxisEncoderOffset;
			st_drive_cmd.enu_cmd := READ_NC_PARAMETER;
		END_IF

		(*-----------------------Weiterschaltbedingungen----------------------------*)
		IF st_drive_cmd.enu_cmd = NO_COMMAND THEN
			IF fb_axis.r_wert_nc_read_parameter = gst_datensatz.st_md.st_md_bestueckachse.lr_nullpunktverschiebung THEN
				fb_state_entry.i16_next_step := 2040;	(* Jogbetrieb *)
			ELSE
				fb_state_entry.i16_next_step := 2010;	(* Reglerfreigabe nehmen und Nullpunktverschiebung schreiben *)
			END_IF
		END_IF

(*=======================================================*)
	2010:	(* Reglerfreigabe wegnehmen , damit Nullpunktverschiebung geschrieben werden kannt*)
		IF fb_state_entry.E THEN
			st_drive_cmd.enu_cmd := POWER_DISABLE;
		END_IF

		(*-----------------------Weiterschaltbedingungen----------------------------*)
		IF st_drive_cmd.enu_cmd = NO_COMMAND THEN
			fb_state_entry.i16_next_step := 2020;
		END_IF

(*=======================================================*)
	2020:	(* Nullpunktverschiebung hat sich geändert, deshalb erst Null reinschreiben, um keinen Additionsfehler zu machen, *)
			(* weil der Wert der Verschiebung beim Neustart komplett auf die Achse geschrieben wird *)
		IF fb_state_entry.E THEN
			fb_axis.i16_nc_parameter_nummer := AxisEncoderOffset;
			fb_axis.r_wert_nc_write_parameter := 0.0;
			st_drive_cmd.enu_cmd := WRITE_NC_PARAMETER;
		END_IF

		(*-----------------------Weiterschaltbedingungen----------------------------*)
		IF st_drive_cmd.enu_cmd = NO_COMMAND THEN
			fb_state_entry.i16_next_step := 2030;
		END_IF

(*=======================================================*)
	2030:	(* Aktuelle Nullpunktverschiebung des Absolutwertgebers an die Achse senden *)
		IF fb_state_entry.E THEN
			fb_axis.i16_nc_parameter_nummer := AxisEncoderOffset;
			fb_axis.r_wert_nc_write_parameter := gst_datensatz.st_md.st_md_bestueckachse.lr_nullpunktverschiebung;
			st_drive_cmd.enu_cmd := WRITE_NC_PARAMETER;
		END_IF

		(*-----------------------Weiterschaltbedingungen----------------------------*)
		IF st_drive_cmd.enu_cmd = NO_COMMAND THEN
			fb_state_entry.i16_next_step := 2040;
		END_IF

(*=======================================================*)
	2040:	(* Jogbetrieb *)
		IF fb_state_entry.E THEN
			fb_axis.lr_soll_geschwindigkeit := st_geschwindigkeiten.lr_jog;
		END_IF

		IF ST_Euchner_Handbedienpult.i16_Handrad_delta > 0 THEN
			st_drive_cmd.enu_cmd := JOG_VORWAERTS;
		ELSIF ST_Euchner_Handbedienpult.i16_Handrad_delta < 0 THEN
			st_drive_cmd.enu_cmd := JOG_RUECKWAERTS;
		ELSE
			IF bestueckachse.Status.Moving THEN
				st_drive_cmd.enu_cmd := JOG_STOP;
			END_IF
		END_IF

		IF fb_r_trig_taste_plus.Q THEN
			fb_state_entry.i16_next_step := MOTORBREMSE_AUF;
		END_IF
		IF fb_r_trig_taste_minus.Q THEN
			fb_state_entry.i16_next_step := MOTORBREMSE_ZU;
		END_IF

		(*-----------------------Weiterschaltbedingungen----------------------------*)
		IF gi16_betriebsart <> HAND OR NOT b_hand_dialog_aktiv THEN
			fb_state_entry.i16_next_step := 2050;
		END_IF

(*=======================================================*)
	2050:
		IF fb_state_entry.E THEN
			st_drive_cmd.enu_cmd := ABORT;
		END_IF

		(*-----------------------Weiterschaltbedingungen----------------------------*)
		IF st_drive_cmd.enu_cmd = NO_COMMAND THEN
			fb_state_entry.i16_next_step := 2060;
		END_IF

(*=======================================================*)
	2060:
		IF fb_state_entry.E THEN
			fb_axis.w_idn := P_0_IDN + 96;
			fb_axis.ui16_soeparam_write_value := 0;	(* Motorbremse im Automatikbetrieb für reguläres Fahren *)
			st_drive_cmd.enu_cmd := SOE_WRITE_PARAM;
		END_IF

		(*-----------------------Weiterschaltbedingungen----------------------------*)
		IF st_drive_cmd.enu_cmd = NO_COMMAND THEN
			fb_state_entry.i16_next_step := 2070;
		END_IF

(*=======================================================*)
	2070:	(* Reglerfreigabe wegnehmen *)
		IF fb_state_entry.E THEN
			st_drive_cmd.enu_cmd := POWER_DISABLE;
		END_IF

		(*-----------------------Weiterschaltbedingungen----------------------------*)
		IF st_drive_cmd.enu_cmd = NO_COMMAND THEN
			st_ctrl_out.b_fehler := FALSE;
			fb_state_entry.i16_next_step := INIT;
		END_IF

(*=======================================================*)
	MOTORBREMSE_AUF:
		IF fb_state_entry.E THEN
			st_drive_cmd.enu_cmd := ABORT;
		END_IF

		(*-----------------------Weiterschaltbedingungen----------------------------*)
		IF st_drive_cmd.enu_cmd = NO_COMMAND THEN
			fb_state_entry.i16_next_step := 2110;
		END_IF

(*=======================================================*)
	2110:	(* Reglerfreigabe wegnehmen *)
		IF fb_state_entry.E THEN
			st_drive_cmd.enu_cmd := POWER_DISABLE;
		END_IF

		(*-----------------------Weiterschaltbedingungen----------------------------*)
		IF st_drive_cmd.enu_cmd = NO_COMMAND THEN
			fb_state_entry.i16_next_step := 2120;
		END_IF

(*=======================================================*)
	2120:	(* Bremse auf machen *)
		IF fb_state_entry.E THEN
			fb_axis.w_idn := P_0_IDN + 96;
			fb_axis.ui16_soeparam_write_value := 2;
			st_drive_cmd.enu_cmd := SOE_WRITE_PARAM;
		END_IF

		(*-----------------------Weiterschaltbedingungen----------------------------*)
		IF 	st_drive_cmd.enu_cmd = NO_COMMAND AND
			(gi16_betriebsart <> HAND OR
			NOT b_hand_dialog_aktiv OR
			ST_Euchner_Handbedienpult.i16_Handrad_delta > 0)
			THEN
				fb_state_entry.i16_next_step := HANDRAD;
		ELSIF fb_r_trig_taste_minus.Q THEN
			fb_state_entry.i16_next_step := MOTORBREMSE_ZU;
		END_IF

(*=======================================================*)
	MOTORBREMSE_ZU:
		IF fb_state_entry.E THEN
			st_drive_cmd.enu_cmd := ABORT;
		END_IF

		(*-----------------------Weiterschaltbedingungen----------------------------*)
		IF st_drive_cmd.enu_cmd = NO_COMMAND THEN
			fb_state_entry.i16_next_step := 2210;
		END_IF

(*=======================================================*)
	2210:	(* Reglerfreigabe setzen *)
		IF fb_state_entry.E THEN
			st_drive_cmd.enu_cmd := POWER_ENABLE;
		END_IF

		(*-----------------------Weiterschaltbedingungen----------------------------*)
		IF st_drive_cmd.enu_cmd = NO_COMMAND THEN
			fb_state_entry.i16_next_step := 2220;
		END_IF

(*=======================================================*)
	2220:	(* Bremse zu machen *)
		IF fb_state_entry.E THEN
			fb_axis.w_idn := P_0_IDN + 96;
			fb_axis.ui16_soeparam_write_value := 0;	(* Motorbremse im Automatikbetrieb für reguläres Fahren *)
			st_drive_cmd.enu_cmd := SOE_WRITE_PARAM;
		END_IF

		(*-----------------------Weiterschaltbedingungen----------------------------*)
		IF 	st_drive_cmd.enu_cmd = NO_COMMAND AND
			(gi16_betriebsart <> HAND OR
			NOT b_hand_dialog_aktiv OR
			ST_Euchner_Handbedienpult.i16_Handrad_delta > 0)
			THEN
				fb_state_entry.i16_next_step := HANDRAD;
		ELSIF fb_r_trig_taste_plus.Q THEN
			fb_state_entry.i16_next_step := MOTORBREMSE_AUF;
		END_IF

(*=======================================================*)
	NULLPUNKT_SETZEN:
		(* Aktuellen Jog beenden, sonst Probleme beim Softwareendschalter*)
		IF fb_state_entry.E THEN
			st_drive_cmd.enu_cmd := JOG_STOP;
		END_IF

		(*-----------------------Weiterschaltbedingungen----------------------------*)
		IF st_drive_cmd.enu_cmd = NO_COMMAND THEN
			fb_state_entry.i16_next_step := 2505;
		END_IF

(*=======================================================*)
	2505:
		(* 	Lese aktuelle Nullpunkt verschiebung von der Hardware. Der Benutze könnte einen falschen
			Wert eingetragen haben *)
		IF fb_state_entry.E THEN
			fb_axis.i16_nc_parameter_nummer := AxisEncoderOffset;
			st_drive_cmd.enu_cmd := READ_NC_PARAMETER;
		END_IF

		(*-----------------------Weiterschaltbedingungen----------------------------*)
		IF st_drive_cmd.enu_cmd = NO_COMMAND THEN
			gst_datensatz.st_md.st_md_bestueckachse.lr_nullpunktverschiebung := fb_axis.r_wert_nc_read_parameter;
			fb_state_entry.i16_next_step := 2510;
		END_IF

(*=======================================================*)
	2510:	(* Nullpunktverschiebung berechnen *)
		IF fb_state_entry.E THEN
			lr_pos_ohneverschiebung := axis_bestueckachse.st_visu.lr_position_ist - gst_datensatz.st_md.st_md_bestueckachse.lr_nullpunktverschiebung;
		
			gst_datensatz.st_md.st_md_bestueckachse.lr_nullpunktverschiebung := - lr_pos_ohneverschiebung;
	
			WHILE (gst_datensatz.st_md.st_md_bestueckachse.lr_nullpunktverschiebung > 360)
			DO
				gst_datensatz.st_md.st_md_bestueckachse.lr_nullpunktverschiebung :=
					gst_datensatz.st_md.st_md_bestueckachse.lr_nullpunktverschiebung - 360;
			END_WHILE
		
			WHILE (gst_datensatz.st_md.st_md_bestueckachse.lr_nullpunktverschiebung < 0)
			DO
				gst_datensatz.st_md.st_md_bestueckachse.lr_nullpunktverschiebung :=
					gst_datensatz.st_md.st_md_bestueckachse.lr_nullpunktverschiebung + 360;
			END_WHILE
		END_IF

		(*-----------------------Weiterschaltbedingungen----------------------------*)
		(* Aktiviere den wert in die Hardware *)
		fb_state_entry.i16_next_step := HANDRAD;

(*=======================================================*)
	INBETRIEBNAHME:	(* Überprüfe Nullpunktverschiebung des Absolutwertgebers auf Korrektheit *)
		IF fb_state_entry.E THEN
			fb_axis.i16_nc_parameter_nummer := AxisEncoderOffset;
			st_drive_cmd.enu_cmd := READ_NC_PARAMETER;
		END_IF

		(*-----------------------Weiterschaltbedingungen----------------------------*)
		IF st_drive_cmd.enu_cmd = NO_COMMAND THEN
			IF fb_axis.r_wert_nc_read_parameter = gst_datensatz.st_md.st_md_bestueckachse.lr_nullpunktverschiebung THEN
				fb_state_entry.i16_next_step := 5100;	(* Reversiersequenz*)
			ELSE
				fb_state_entry.i16_next_step := 5010;	(* Reglerfreigabe nehmen und Nullpunktverschiebung schreiben *)
			END_IF
		END_IF

(*=======================================================*)
	5010:	(* Reglerfreigabe wegnehmen, damit Nullpunktverschiebung geschrieben werden kannt*)
		IF fb_state_entry.E THEN
			st_drive_cmd.enu_cmd := POWER_DISABLE;
		END_IF

		(*-----------------------Weiterschaltbedingungen----------------------------*)
		IF st_drive_cmd.enu_cmd = NO_COMMAND THEN
			fb_state_entry.i16_next_step := 5020;
		END_IF

(*=======================================================*)
	5020:	(* Nullpunktverschiebung hat sich geändert, deshalb erst Null reinschreiben, um keinen Additionsfehler zu machen, *)
			(* weil der Wert der Verschiebung beim Neustart komplett auf die Achse geschrieben wird *)
		IF fb_state_entry.E THEN
			fb_axis.i16_nc_parameter_nummer := AxisEncoderOffset;
			fb_axis.r_wert_nc_write_parameter := 0.0;
			st_drive_cmd.enu_cmd := WRITE_NC_PARAMETER;
		END_IF

		(*-----------------------Weiterschaltbedingungen----------------------------*)
		IF st_drive_cmd.enu_cmd = NO_COMMAND THEN
			fb_state_entry.i16_next_step := 5030;
		END_IF

(*=======================================================*)
	5030:	(* Aktuelle Nullpunktverschiebung des Absolutwertgebers an die Achse senden *)
		IF fb_state_entry.E THEN
			fb_axis.i16_nc_parameter_nummer := AxisEncoderOffset;
			fb_axis.r_wert_nc_write_parameter := gst_datensatz.st_md.st_md_bestueckachse.lr_nullpunktverschiebung;
			st_drive_cmd.enu_cmd := WRITE_NC_PARAMETER;
		END_IF

		(*-----------------------Weiterschaltbedingungen----------------------------*)
		IF st_drive_cmd.enu_cmd = NO_COMMAND THEN
			fb_state_entry.i16_next_step := 5100;
		END_IF

(*=======================================================*)
	5100:	(* Verfahren der Achse zwischen zwei Punkten zum Testen verschiedener Achsparameter *)
		IF fb_state_entry.E THEN
			fb_axis.lr_soll_geschwindigkeit := st_geschwindigkeiten.lr_jog;
			fb_axis.st_position.lr_ibn_pos_start := 0.0;
			fb_axis.st_position.lr_ibn_pos_ziel := 180.0;
		END_IF

		(*-----------------------Weiterschaltbedingungen----------------------------*)
		IF st_ctrl_in.b_ibn_start THEN
			fb_state_entry.i16_next_step := 5110;
		END_IF

(*=======================================================*)
	5110: (* Fahre Bestückachse auf Startposition *)
(*
		IF fb_state_entry.E THEN
			 fb_axis.st_position.r_soll := fb_axis.st_position.lr_ibn_pos_start;
			fb_axis.mc_richtung_modulo :=MC_Positive_Direction ;
			st_drive_cmd.enu_cmd := MOVE_MODULO;
		END_IF

		(*-----------------------Weiterschaltbedingungen----------------------------*)
		IF st_drive_cmd.enu_cmd = NO_COMMAND THEN
			fb_state_entry.i16_next_step := 5120;
		END_IF
*)
		IF fb_state_entry.E THEN
			st_drive_cmd.enu_cmd := POWER_ENABLE;
		END_IF

		(*-----------------------Weiterschaltbedingungen----------------------------*)
		IF st_drive_cmd.enu_cmd = NO_COMMAND THEN
			;
		END_IF

(*=======================================================*)
	5120: (* Pause *)
		IF fb_state_entry.E THEN
			fb_ton_wz.PT := t#1s;
			fb_ton_wz.IN := TRUE;
		END_IF

		(*-----------------------Weiterschaltbedingungen----------------------------*)
		IF fb_ton_wz.Q THEN
			fb_ton_wz.IN := FALSE;
			fb_state_entry.i16_next_step := 5130;
		END_IF

(*=======================================================*)
	5130: (* Fahre Bestückachse auf Zielposition *)
		IF fb_state_entry.E THEN
			 fb_axis.st_position.r_soll := fb_axis.st_position.lr_ibn_pos_ziel;
			fb_axis.mc_richtung_modulo :=MC_Negative_Direction ;
			st_drive_cmd.enu_cmd := MOVE_MODULO;
		END_IF

		(*-----------------------Weiterschaltbedingungen----------------------------*)
		IF st_drive_cmd.enu_cmd = NO_COMMAND THEN
			fb_state_entry.i16_next_step := 5140;
		END_IF

(*=======================================================*)
	5140: (* Pause *)
		IF fb_state_entry.E THEN
			fb_ton_wz.PT := t#1s;
			fb_ton_wz.IN := TRUE;
		END_IF

		(*-----------------------Weiterschaltbedingungen----------------------------*)
		IF fb_ton_wz.Q THEN
			fb_ton_wz.IN := FALSE;
			fb_state_entry.i16_next_step := 5100;
		END_IF
END_CASE

fb_state_entry(
	i16_next_step:= , 
	i16_pos:= 2,
	s_debugtext:= ,
	E=> ,
	X=> ,
	i16_step=> ,
	i16_last_step=> );

IF st_config_achse.b_config_fertig THEN
	(* Fehlermeldungen und Betriebsmeldungen ab dem Startindex in die globalen Meldungsarrays schreiben *)
	garr_stoermeldungen[st_config_achse.i16_meld_startindex + 0] := st_sm.b_achse_nicht_bb;
	garr_stoermeldungen[st_config_achse.i16_meld_startindex + 1] := st_sm.b_achse_nicht_referenziert;
	garr_stoermeldungen[st_config_achse.i16_meld_startindex + 2] := st_sm.b_keine_verfahrfreigabe;
	garr_stoermeldungen[st_config_achse.i16_meld_startindex + 3] := st_sm.b_achse_nicht_auf_startpos;
	garr_stoermeldungen[st_config_achse.i16_meld_startindex + 4] := st_sm.b_ende_skalierungs_nocke;
	garr_stoermeldungen[st_config_achse.i16_meld_startindex + 5] := st_sm.b_ende_camming_nocke;
	garr_stoermeldungen[st_config_achse.i16_meld_startindex + 6] := st_sm.b_skalierung_noch_aktiv;
	garr_stoermeldungen[st_config_achse.i16_meld_startindex + 7] := FALSE;
	garr_stoermeldungen[st_config_achse.i16_meld_startindex + 8] := FALSE;
	garr_stoermeldungen[st_config_achse.i16_meld_startindex + 9] := FALSE;
	garr_stoermeldungen[st_config_achse.i16_meld_startindex + 10] := FALSE;
	garr_stoermeldungen[st_config_achse.i16_meld_startindex + 11] := FALSE;
	garr_stoermeldungen[st_config_achse.i16_meld_startindex + 12] := sm_fehler_initialposition_achse;
	garr_stoermeldungen[st_config_achse.i16_meld_startindex + 13] := sm_keine_nocken_definiert;
	garr_stoermeldungen[st_config_achse.i16_meld_startindex + 14] := FALSE;
	garr_stoermeldungen[st_config_achse.i16_meld_startindex + 15] := sm_fehler_ot_ut;
	garr_stoermeldungen[st_config_achse.i16_meld_startindex + 16] := st_drive_cmd.meldungen.sm_write_soe_parameter;
	garr_stoermeldungen[st_config_achse.i16_meld_startindex + 17] := st_drive_cmd.meldungen.sm_read_soe_parameter;
	garr_stoermeldungen[st_config_achse.i16_meld_startindex + 18] := st_drive_cmd.meldungen.sm_write_nc_parameter;
	garr_stoermeldungen[st_config_achse.i16_meld_startindex + 19] := st_drive_cmd.meldungen.sm_read_nc_parameter;
	garr_stoermeldungen[st_config_achse.i16_meld_startindex + 20] := st_drive_cmd.meldungen.sm_power_enable;
	garr_stoermeldungen[st_config_achse.i16_meld_startindex + 21] := st_drive_cmd.meldungen.sm_power_disable;
	garr_stoermeldungen[st_config_achse.i16_meld_startindex + 22] := st_drive_cmd.meldungen.sm_reset;
	garr_stoermeldungen[st_config_achse.i16_meld_startindex + 23] := st_drive_cmd.meldungen.sm_home;
	garr_stoermeldungen[st_config_achse.i16_meld_startindex + 24] := st_drive_cmd.meldungen.sm_setposition;
	garr_stoermeldungen[st_config_achse.i16_meld_startindex + 25] := st_drive_cmd.meldungen.sm_jog_vorwaerts;
	garr_stoermeldungen[st_config_achse.i16_meld_startindex + 26] := st_drive_cmd.meldungen.sm_jog_rueckwaerts;
	garr_stoermeldungen[st_config_achse.i16_meld_startindex + 27] := st_drive_cmd.meldungen.sm_move_absolute;
	garr_stoermeldungen[st_config_achse.i16_meld_startindex + 28] := st_drive_cmd.meldungen.sm_move_relative;
	garr_stoermeldungen[st_config_achse.i16_meld_startindex + 29] := st_drive_cmd.meldungen.sm_move_velocity;
	garr_stoermeldungen[st_config_achse.i16_meld_startindex + 30] := st_drive_cmd.meldungen.sm_move_modulo;
	garr_stoermeldungen[st_config_achse.i16_meld_startindex + 31] := st_drive_cmd.meldungen.sm_stop_axis;
	garr_stoermeldungen[st_config_achse.i16_meld_startindex + 32] := st_drive_cmd.meldungen.sm_halt_axis;
	garr_stoermeldungen[st_config_achse.i16_meld_startindex + 33] := st_drive_cmd.meldungen.sm_motion_command_timeout;
	garr_stoermeldungen[st_config_achse.i16_meld_startindex + 34] := st_sm.b_achsfehler;
	garr_stoermeldungen[st_config_achse.i16_meld_startindex + 35] := st_sm.b_devicefehler;
	garr_stoermeldungen[st_config_achse.i16_meld_startindex + 36] := st_drive_cmd.meldungen.sm_limit_positiv_erreicht;
	garr_stoermeldungen[st_config_achse.i16_meld_startindex + 37] := st_drive_cmd.meldungen.sm_limit_negativ_erreicht;
	garr_stoermeldungen[st_config_achse.i16_meld_startindex + 38] := st_drive_cmd.meldungen.sm_ec_coe_sdo_write_ex;
	garr_stoermeldungen[st_config_achse.i16_meld_startindex + 39] := st_drive_cmd.meldungen.sm_ec_coe_sdo_read_ex;
	garr_stoermeldungen[st_config_achse.i16_meld_startindex + 40] := FALSE;
	garr_stoermeldungen[st_config_achse.i16_meld_startindex + 41] := FALSE;
	garr_stoermeldungen[st_config_achse.i16_meld_startindex + 42] := FALSE;
	garr_stoermeldungen[st_config_achse.i16_meld_startindex + 43] := FALSE;
	garr_stoermeldungen[st_config_achse.i16_meld_startindex + 44] := FALSE;
	garr_stoermeldungen[st_config_achse.i16_meld_startindex + 45] := FALSE;
	garr_stoermeldungen[st_config_achse.i16_meld_startindex + 46] := FALSE;
	garr_stoermeldungen[st_config_achse.i16_meld_startindex + 47] := FALSE;
	garr_stoermeldungen[st_config_achse.i16_meld_startindex + 48] := FALSE;
	garr_stoermeldungen[st_config_achse.i16_meld_startindex + 49] := FALSE;
	garr_stoermeldungen[st_config_achse.i16_meld_startindex + 50] := FALSE;
	garr_stoermeldungen[st_config_achse.i16_meld_startindex + 51] := FALSE;
	garr_stoermeldungen[st_config_achse.i16_meld_startindex + 52] := FALSE;
	garr_stoermeldungen[st_config_achse.i16_meld_startindex + 53] := FALSE;
	garr_stoermeldungen[st_config_achse.i16_meld_startindex + 54] := FALSE;
	garr_stoermeldungen[st_config_achse.i16_meld_startindex + 55] := FALSE;
	garr_stoermeldungen[st_config_achse.i16_meld_startindex + 56] := FALSE;
	garr_stoermeldungen[st_config_achse.i16_meld_startindex + 57] := FALSE;
	garr_stoermeldungen[st_config_achse.i16_meld_startindex + 58] := FALSE;
	garr_stoermeldungen[st_config_achse.i16_meld_startindex + 59] := FALSE;
	garr_stoermeldungen[st_config_achse.i16_meld_startindex + 60] := FALSE;
	garr_stoermeldungen[st_config_achse.i16_meld_startindex + 61] := FALSE;
	garr_stoermeldungen[st_config_achse.i16_meld_startindex + 62] := FALSE;
	garr_stoermeldungen[st_config_achse.i16_meld_startindex + 63] := FALSE;
	garr_stoermeldungen[st_config_achse.i16_meld_startindex + 64] := FALSE;
	garr_stoermeldungen[st_config_achse.i16_meld_startindex + 65] := FALSE;
	garr_stoermeldungen[st_config_achse.i16_meld_startindex + 66] := FALSE;
	garr_stoermeldungen[st_config_achse.i16_meld_startindex + 67] := FALSE;
	garr_stoermeldungen[st_config_achse.i16_meld_startindex + 68] := FALSE;
	garr_stoermeldungen[st_config_achse.i16_meld_startindex + 69] := FALSE;
	garr_stoermeldungen[st_config_achse.i16_meld_startindex + 70] :=  FALSE;
	garr_stoermeldungen[st_config_achse.i16_meld_startindex + 71] :=  FALSE;
	garr_stoermeldungen[st_config_achse.i16_meld_startindex + 72] :=  FALSE;
	garr_stoermeldungen[st_config_achse.i16_meld_startindex + 73] :=  FALSE;
	garr_stoermeldungen[st_config_achse.i16_meld_startindex + 74] :=  FALSE;
	garr_stoermeldungen[st_config_achse.i16_meld_startindex + 75] :=  FALSE;
	garr_stoermeldungen[st_config_achse.i16_meld_startindex + 76] :=  FALSE;
	garr_stoermeldungen[st_config_achse.i16_meld_startindex + 77] :=  FALSE;
	garr_stoermeldungen[st_config_achse.i16_meld_startindex + 78] :=  FALSE;
	garr_stoermeldungen[st_config_achse.i16_meld_startindex + 79] :=  FALSE;
	garr_stoermeldungen[st_config_achse.i16_meld_startindex + 80] :=  FALSE;
	garr_stoermeldungen[st_config_achse.i16_meld_startindex + 81] :=  FALSE;
	garr_stoermeldungen[st_config_achse.i16_meld_startindex + 82] :=  FALSE;
	garr_stoermeldungen[st_config_achse.i16_meld_startindex + 83] :=  FALSE;
	garr_stoermeldungen[st_config_achse.i16_meld_startindex + 84] :=  FALSE;
	garr_stoermeldungen[st_config_achse.i16_meld_startindex + 85] :=  FALSE;
	garr_stoermeldungen[st_config_achse.i16_meld_startindex + 86] :=  FALSE;
	garr_stoermeldungen[st_config_achse.i16_meld_startindex + 87] :=  FALSE;
	garr_stoermeldungen[st_config_achse.i16_meld_startindex + 88] :=  FALSE;
	garr_stoermeldungen[st_config_achse.i16_meld_startindex + 89] :=  FALSE;
	garr_stoermeldungen[st_config_achse.i16_meld_startindex + 90] :=  FALSE;
	garr_stoermeldungen[st_config_achse.i16_meld_startindex + 91] :=  FALSE;
	garr_stoermeldungen[st_config_achse.i16_meld_startindex + 92] :=  FALSE;
	garr_stoermeldungen[st_config_achse.i16_meld_startindex + 93] :=  FALSE;
	garr_stoermeldungen[st_config_achse.i16_meld_startindex + 94] :=  FALSE;
	garr_stoermeldungen[st_config_achse.i16_meld_startindex + 95] :=  FALSE;
	garr_stoermeldungen[st_config_achse.i16_meld_startindex + 96] :=  FALSE;
	garr_stoermeldungen[st_config_achse.i16_meld_startindex + 97] :=  FALSE;
	garr_stoermeldungen[st_config_achse.i16_meld_startindex + 98] :=  FALSE;
	garr_stoermeldungen[st_config_achse.i16_meld_startindex + 99] :=  FALSE;

	garr_betriebsmeldungen[st_config_achse.i16_meld_startindex + 0] := FALSE;
	garr_betriebsmeldungen[st_config_achse.i16_meld_startindex + 1] := FALSE;
	garr_betriebsmeldungen[st_config_achse.i16_meld_startindex + 2] := FALSE;
	garr_betriebsmeldungen[st_config_achse.i16_meld_startindex + 3] := FALSE;
	garr_betriebsmeldungen[st_config_achse.i16_meld_startindex + 4] := FALSE;
	garr_betriebsmeldungen[st_config_achse.i16_meld_startindex + 5] := FALSE;
	garr_betriebsmeldungen[st_config_achse.i16_meld_startindex + 6] := FALSE;
	garr_betriebsmeldungen[st_config_achse.i16_meld_startindex + 7] := FALSE;
	garr_betriebsmeldungen[st_config_achse.i16_meld_startindex + 8] := FALSE;
	garr_betriebsmeldungen[st_config_achse.i16_meld_startindex + 9] := FALSE;
	garr_betriebsmeldungen[st_config_achse.i16_meld_startindex + 10] := FALSE;
	garr_betriebsmeldungen[st_config_achse.i16_meld_startindex + 11] := FALSE;
	garr_betriebsmeldungen[st_config_achse.i16_meld_startindex + 12] := FALSE;
	garr_betriebsmeldungen[st_config_achse.i16_meld_startindex + 13] := FALSE;
	garr_betriebsmeldungen[st_config_achse.i16_meld_startindex + 14] := FALSE;
	garr_betriebsmeldungen[st_config_achse.i16_meld_startindex + 15] := FALSE;
	garr_betriebsmeldungen[st_config_achse.i16_meld_startindex + 16] := FALSE;
	garr_betriebsmeldungen[st_config_achse.i16_meld_startindex + 17] := FALSE;
	garr_betriebsmeldungen[st_config_achse.i16_meld_startindex + 18] := FALSE;
	garr_betriebsmeldungen[st_config_achse.i16_meld_startindex + 19] := FALSE;
	garr_betriebsmeldungen[st_config_achse.i16_meld_startindex + 20] := FALSE;
	garr_betriebsmeldungen[st_config_achse.i16_meld_startindex + 21] := FALSE;
	garr_betriebsmeldungen[st_config_achse.i16_meld_startindex + 22] := FALSE;
	garr_betriebsmeldungen[st_config_achse.i16_meld_startindex + 23] := FALSE;
	garr_betriebsmeldungen[st_config_achse.i16_meld_startindex + 24] := FALSE;
	garr_betriebsmeldungen[st_config_achse.i16_meld_startindex + 25] := FALSE;
	garr_betriebsmeldungen[st_config_achse.i16_meld_startindex + 26] := FALSE;
	garr_betriebsmeldungen[st_config_achse.i16_meld_startindex + 27] := FALSE;
	garr_betriebsmeldungen[st_config_achse.i16_meld_startindex + 28] := FALSE;
	garr_betriebsmeldungen[st_config_achse.i16_meld_startindex + 29] := FALSE;
	garr_betriebsmeldungen[st_config_achse.i16_meld_startindex + 30] := FALSE;
	garr_betriebsmeldungen[st_config_achse.i16_meld_startindex + 31] := FALSE;
	garr_betriebsmeldungen[st_config_achse.i16_meld_startindex + 32] := FALSE;
	garr_betriebsmeldungen[st_config_achse.i16_meld_startindex + 33] := FALSE;
	garr_betriebsmeldungen[st_config_achse.i16_meld_startindex + 34] := FALSE;
	garr_betriebsmeldungen[st_config_achse.i16_meld_startindex + 35] := FALSE;
	garr_betriebsmeldungen[st_config_achse.i16_meld_startindex + 36] := FALSE;
	garr_betriebsmeldungen[st_config_achse.i16_meld_startindex + 37] := FALSE;
	garr_betriebsmeldungen[st_config_achse.i16_meld_startindex + 38] := FALSE;
	garr_betriebsmeldungen[st_config_achse.i16_meld_startindex + 39] := FALSE;
	garr_betriebsmeldungen[st_config_achse.i16_meld_startindex + 40] := FALSE;
	garr_betriebsmeldungen[st_config_achse.i16_meld_startindex + 41] := FALSE;
	garr_betriebsmeldungen[st_config_achse.i16_meld_startindex + 42] := FALSE;
	garr_betriebsmeldungen[st_config_achse.i16_meld_startindex + 43] := FALSE;
	garr_betriebsmeldungen[st_config_achse.i16_meld_startindex + 44] := FALSE;
	garr_betriebsmeldungen[st_config_achse.i16_meld_startindex + 45] := FALSE;
	garr_betriebsmeldungen[st_config_achse.i16_meld_startindex + 46] := FALSE;
	garr_betriebsmeldungen[st_config_achse.i16_meld_startindex + 47] := FALSE;
	garr_betriebsmeldungen[st_config_achse.i16_meld_startindex + 48] := FALSE;
	garr_betriebsmeldungen[st_config_achse.i16_meld_startindex + 49] := FALSE;
	garr_betriebsmeldungen[st_config_achse.i16_meld_startindex + 50] := FALSE;
	garr_betriebsmeldungen[st_config_achse.i16_meld_startindex + 51] := FALSE;
	garr_betriebsmeldungen[st_config_achse.i16_meld_startindex + 52] := FALSE;
	garr_betriebsmeldungen[st_config_achse.i16_meld_startindex + 53] := FALSE;
	garr_betriebsmeldungen[st_config_achse.i16_meld_startindex + 54] := FALSE;
	garr_betriebsmeldungen[st_config_achse.i16_meld_startindex + 55] := FALSE;
	garr_betriebsmeldungen[st_config_achse.i16_meld_startindex + 56] := FALSE;
	garr_betriebsmeldungen[st_config_achse.i16_meld_startindex + 57] := FALSE;
	garr_betriebsmeldungen[st_config_achse.i16_meld_startindex + 58] := FALSE;
	garr_betriebsmeldungen[st_config_achse.i16_meld_startindex + 59] := FALSE;
	garr_betriebsmeldungen[st_config_achse.i16_meld_startindex + 60] := FALSE;
	garr_betriebsmeldungen[st_config_achse.i16_meld_startindex + 61] := FALSE;
	garr_betriebsmeldungen[st_config_achse.i16_meld_startindex + 62] := FALSE;
	garr_betriebsmeldungen[st_config_achse.i16_meld_startindex + 63] := FALSE;
	garr_betriebsmeldungen[st_config_achse.i16_meld_startindex + 64] := FALSE;
	garr_betriebsmeldungen[st_config_achse.i16_meld_startindex + 65] := FALSE;
	garr_betriebsmeldungen[st_config_achse.i16_meld_startindex + 66] := FALSE;
	garr_betriebsmeldungen[st_config_achse.i16_meld_startindex + 67] := FALSE;
	garr_betriebsmeldungen[st_config_achse.i16_meld_startindex + 68] := FALSE;
	garr_betriebsmeldungen[st_config_achse.i16_meld_startindex + 69] := FALSE;
	garr_betriebsmeldungen[st_config_achse.i16_meld_startindex + 70] :=  FALSE;
	garr_betriebsmeldungen[st_config_achse.i16_meld_startindex + 71] :=  FALSE;
	garr_betriebsmeldungen[st_config_achse.i16_meld_startindex + 72] :=  FALSE;
	garr_betriebsmeldungen[st_config_achse.i16_meld_startindex + 73] :=  FALSE;
	garr_betriebsmeldungen[st_config_achse.i16_meld_startindex + 74] :=  FALSE;
	garr_betriebsmeldungen[st_config_achse.i16_meld_startindex + 75] :=  FALSE;
	garr_betriebsmeldungen[st_config_achse.i16_meld_startindex + 76] :=  FALSE;
	garr_betriebsmeldungen[st_config_achse.i16_meld_startindex + 77] :=  FALSE;
	garr_betriebsmeldungen[st_config_achse.i16_meld_startindex + 78] :=  FALSE;
	garr_betriebsmeldungen[st_config_achse.i16_meld_startindex + 79] :=  FALSE;
	garr_betriebsmeldungen[st_config_achse.i16_meld_startindex + 80] :=  FALSE;
	garr_betriebsmeldungen[st_config_achse.i16_meld_startindex + 81] :=  FALSE;
	garr_betriebsmeldungen[st_config_achse.i16_meld_startindex + 82] :=  FALSE;
	garr_betriebsmeldungen[st_config_achse.i16_meld_startindex + 83] :=  FALSE;
	garr_betriebsmeldungen[st_config_achse.i16_meld_startindex + 84] :=  FALSE;
	garr_betriebsmeldungen[st_config_achse.i16_meld_startindex + 85] :=  FALSE;
	garr_betriebsmeldungen[st_config_achse.i16_meld_startindex + 86] :=  FALSE;
	garr_betriebsmeldungen[st_config_achse.i16_meld_startindex + 87] :=  FALSE;
	garr_betriebsmeldungen[st_config_achse.i16_meld_startindex + 88] :=  FALSE;
	garr_betriebsmeldungen[st_config_achse.i16_meld_startindex + 89] :=  FALSE;
	garr_betriebsmeldungen[st_config_achse.i16_meld_startindex + 90] :=  FALSE;
	garr_betriebsmeldungen[st_config_achse.i16_meld_startindex + 91] :=  FALSE;
	garr_betriebsmeldungen[st_config_achse.i16_meld_startindex + 92] :=  FALSE;
	garr_betriebsmeldungen[st_config_achse.i16_meld_startindex + 93] :=  FALSE;
	garr_betriebsmeldungen[st_config_achse.i16_meld_startindex + 94] :=  FALSE;
	garr_betriebsmeldungen[st_config_achse.i16_meld_startindex + 95] :=  FALSE;
	garr_betriebsmeldungen[st_config_achse.i16_meld_startindex + 96] :=  FALSE;
	garr_betriebsmeldungen[st_config_achse.i16_meld_startindex + 97] :=  FALSE;
	garr_betriebsmeldungen[st_config_achse.i16_meld_startindex + 98] :=  FALSE;
	garr_betriebsmeldungen[st_config_achse.i16_meld_startindex + 99] :=  FALSE;
END_IF
END_PROGRAM

(* POU EPT Lib/Funktionsbausteine/ST_OT_UT_Ueberwachung, ST *)
FUNCTION_BLOCK ST_OT_UT_Ueberwachung
VAR_INPUT
	lr_achsposition				 : LREAL;
END_VAR
VAR_OUTPUT
	b_error						: BOOL;
END_VAR
VAR
	i32_anfang_ot					: DINT := 0;
	i32_ende_ot					: DINT := 5;
	i32_anfang_ut					: DINT := 180;
	i32_ende_ut					: DINT := 185;
	arr_eintrag					: ARRAY[0..99] OF BOOL := 1,0,1;	(* Länge dient nur zum Nachverfolgen *)
	b_ot							: BOOL := FALSE;
	b_ut							: BOOL := FALSE;
	fb_r_trig_ot					: R_TRIG;
	fb_r_trig_ut					: R_TRIG;
	fb_f_trig_ot					: F_TRIG;
	fb_f_trig_ut					: F_TRIG;
	i							: INT := 0;
END_VAR
(* Kontrollfunktion zum Prüfen, ob auf OT auch immer UT kommt. *)
(* Die Fehlerausgabe erfolgt mittels temporärer Fehlermeldung, welche im Errorlog der Visu mitgeschrieben wird. *)
(* Dies dient der Kontrolle auf fehlbedienung durch das Anlagenpersonal. *)

(* Flanken *)
fb_r_trig_ot(CLK:= b_ot, Q=> );
fb_r_trig_ut(CLK:= b_ut, Q=> );
fb_f_trig_ot(CLK:= b_ot, Q=> );
fb_f_trig_ut(CLK:= b_ut, Q=> );

(* Erstellen der Bereichsnocken *)
IF LREAL_TO_DINT(lr_achsposition) > i32_anfang_ot AND LREAL_TO_DINT(lr_achsposition) < i32_ende_ot THEN
	b_ot := TRUE;
	b_error := FALSE;
ELSE
	b_ot := FALSE;
END_IF

IF LREAL_TO_DINT(lr_achsposition) > i32_anfang_ut AND LREAL_TO_DINT(lr_achsposition) < i32_ende_ut THEN
	b_ut := TRUE;
	b_error := FALSE;
ELSE
	b_ut := FALSE;
END_IF

(* Eintragen von OT bzw. UT in das Register *)
IF fb_r_trig_ot.Q THEN
	FOR i := 99  TO 1 BY -1 DO
		arr_eintrag [i] := arr_eintrag[i - 1];
	END_FOR
	arr_eintrag[0] := 2#0;	(* Eintrag für OT = 0 *)
END_IF

IF fb_r_trig_ut.Q THEN
	FOR i := 99  TO 1 BY -1 DO
		arr_eintrag[i] := arr_eintrag[i - 1];
	END_FOR
	arr_eintrag[0] := 2#1;	(* Eintrag für UT = 1 *)
END_IF

(* Auswertung und Fehler *)
IF fb_f_trig_ot.Q OR fb_f_trig_ut.Q THEN
	b_error := NOT (arr_eintrag[0]  XOR arr_eintrag[1]);
END_IF
END_FUNCTION_BLOCK

(* POU Maschine1700/Band/ST_Bandwechsel_Kontroller, ST *)
PROGRAM ST_Bandwechsel_Kontroller
VAR_INPUT
	st_config						: struct_config;
	st_ctrl_in						: struct_ctrl_in;
END_VAR
VAR_IN_OUT
	st_visu						: struct_visu;
END_VAR
VAR_OUTPUT
	st_ctrl_out					: struct_ctrl_out;
	b_materialmangel				: BOOL;
	b_materialmangel_links				: BOOL;
	b_materialmangel_rechts				: BOOL;
END_VAR
VAR
	fb_ton_wz					: TON;
	fb_ton_uez					: TON;
	fb_ton_quitt					: TON;
	fb_tof_bandende_li			: TOF;
	fb_tof_bandende_re			: TOF;
	fb_ton_bandende_li			: TON;
	fb_ton_bandende_re			: TON;
	fb_r_trig_start					: R_TRIG;
	fb_r_trig_auto_Bandwechsel_aus: R_TRIG;
	fb_state_entry					: ST_StateEntry;
	b_ibn_start					: BOOL := FALSE;
	fb_r_trig_ibn_start				: R_TRIG;
	fb_ton_ibn_start				: TON;
	i16_vorgabe_einfaedeln		: INT := 0;
	i16_akt_einfaedeln			: INT := 0;
	i16_vorgabe_ausfaedeln		: INT := 0;
	i16_akt_ausfaedeln			: INT := 0;
	i							: INT := 0;
	b_ausgefaedelt				: BOOL;
	b_spulenwechsel				: BOOL;

	sm_halter_nicht_oben			: BOOL:= FALSE;
	sm_bandwechsel_ohne_ende	: BOOL:= FALSE;
	sm_kein_band_anderer_einzug	: BOOL:= FALSE;
	sm_kein_band_in_akt_einzug	: BOOL:= FALSE;
	bm_bandwechselvorgang		: BOOL := FALSE;
	bm_bandwechsel_manuell		: BOOL := FALSE;

	e_ls_bandende_li				AT %I* : BOOL;
	e_ls_bandende_re			AT %I* : BOOL;
END_VAR
(* Zeiten *)
fb_ton_wz(IN:= , PT:= , Q=>  , ET=> );
fb_ton_uez(IN:= , PT:= , Q=>  , ET=> );
fb_ton_quitt(IN:= , PT:= t#100ms, Q=> , ET=> );

fb_ton_bandende_li(IN:= e_ls_bandende_li, PT:= t#1000ms, Q=> , ET=> );
fb_ton_bandende_re(IN:= e_ls_bandende_re, PT:= t#1000ms, Q=> , ET=> );
fb_tof_bandende_li(IN:= fb_ton_bandende_li.Q, PT:= t#1100ms, Q=> , ET=> );
fb_tof_bandende_re(IN:= fb_ton_bandende_re.Q, PT:= t#1100ms, Q=> , ET=> );

(* Flanken *)
fb_r_trig_start(CLK:= st_ctrl_in.b_start, Q=> );

(* Inbetriebnahme *)
fb_r_trig_ibn_start (CLK:= b_ibn_start , Q=> );
fb_ton_ibn_start (IN:= , PT:= t#1s, Q=> , ET=> );

IF fb_r_trig_ibn_start .Q THEN
	fb_ton_ibn_start .IN := TRUE;
ELSE
	IF fb_ton_ibn_start .Q THEN
		b_ibn_start  := FALSE;
	 	fb_ton_ibn_start .IN := FALSE;
	END_IF
END_IF

(* auto Bandwechsel aus *)
fb_r_trig_auto_Bandwechsel_aus(CLK:=visu_hinten.out.auto_Bandwechsel_aus, Q=>);

IF	fb_r_trig_auto_Bandwechsel_aus.Q THEN
	gst_datensatz.st_md.b_auto_Bandwechsel:=NOT gst_datensatz.st_md.b_auto_Bandwechsel;
END_IF
visu_hinten.in.Lampe_auto_Bandwechsel:=gst_datensatz.st_md.b_auto_Bandwechsel;


(* Hier nur Abschaltungen welche zum Bandwechsel Stop führen müssen *)
IF	axis_bestueckachse.st_ctrl.out.b_fehler OR
	axis_z_achse.st_ctrl.out.b_fehler OR
	axis_y_achse.st_ctrl.out.b_fehler OR
	bandspruehoeler.st_ctrl.out.b_fehler OR
	bandeinzug_kontroller.st_ctrl.out.b_fehler OR
	bandwechsel_kontroller.st_ctrl.out.b_fehler OR
	wkz_absicherung.st_ctrl.out.b_fehler OR
	wt_transport_kontroller.st_ctrl.out.b_fehler OR
	hublift_links.st_ctrl.out.b_fehler OR
	hublift_rechts.st_ctrl.out.b_fehler OR
	balluff_tag_reader.st_ctrl.out.b_fehler OR
	haspel_kontroller.st_ctrl.out.b_fehler OR
	bbgen.st_ctrl.out.b_fehler OR
	einpresskraft_kontroller.st_ctrl.out.b_fehler OR
	edit_mfps.st_ctrl.out.b_fehler OR
	Lesen_Schreiben_Tag.st_ctrl.out.b_fehler OR
	Service.st_ctrl.out.b_fehler OR
	gi16_betriebsart = HAND
	THEN
		visu_hinten.in.b_bandwechsel_aktiv := FALSE;
		visu_hinten.in.current_visu_folie := 'BA_1700_BAND_EINFAEDELN';
END_IF

(* Toplevel *)
IF fb_state_entry.i16_step < FEHLER THEN
	IF st_ctrl_in.b_stop THEN
		fb_state_entry.i16_next_step := STOP;
	END_IF
	(* Allgemeine Fehler *)
	IF	NOT gst_datensatz.st_md.b_wt_transport_simulation AND
		(zyl_bawe_vorschub.st_ctrl.out.b_fehler OR
		zyl_bawe_querschub.st_ctrl.out.b_fehler OR
		zyl_bawe_faenger_li.st_ctrl.out.b_fehler OR
		zyl_bawe_faenger_re.st_ctrl.out.b_fehler OR
		zyl_bawe_halter_li.st_ctrl.out.b_fehler OR
		zyl_bawe_halter_re.st_ctrl.out.b_fehler OR
		zyl_haspel_verschieben.st_ctrl.out.b_fehler OR
		zyl_bandeinzuege_verschieben.st_ctrl.out.b_fehler)
		THEN
			fb_state_entry.i16_next_step := FEHLER;
	(* Zylinder im Handbetrieb *)
	ELSIF gi16_betriebsart = HAND AND (
			(st_visu.st_zyl.i16_nr_zyl_im_handbetrieb = zyl_bawe_vorschub.fb.st_config.i16_identnummer) OR
			(st_visu.st_zyl.i16_nr_zyl_im_handbetrieb = zyl_bawe_querschub.fb.st_config.i16_identnummer) OR
			(st_visu.st_zyl.i16_nr_zyl_im_handbetrieb = zyl_bawe_faenger_li.fb.st_config.i16_identnummer) OR
			(st_visu.st_zyl.i16_nr_zyl_im_handbetrieb = zyl_bawe_faenger_re.fb.st_config.i16_identnummer ) OR
			(st_visu.st_zyl.i16_nr_zyl_im_handbetrieb = zyl_bawe_halter_li.fb.st_config.i16_identnummer) OR
			(st_visu.st_zyl.i16_nr_zyl_im_handbetrieb = zyl_bawe_halter_re.fb.st_config.i16_identnummer)OR
			(st_visu.st_zyl.i16_nr_zyl_im_handbetrieb = zyl_haspel_verschieben.fb.st_config.i16_identnummer)OR
			(st_visu.st_zyl.i16_nr_zyl_im_handbetrieb = zyl_bandeinzuege_verschieben.fb.st_config.i16_identnummer))
			THEN
				fb_state_entry.i16_next_step := FEHLER;
	END_IF
END_IF

(* Bandwechsel wird durch eine gelbe Dauerleuchte angezeigt *)
b_materialmangel := b_materialmangel_links OR b_materialmangel_rechts;

IF	b_ausgefaedelt THEN
	IF 	b_materialmangel_links AND
		NOT fb_tof_bandende_li.Q THEN
		b_materialmangel_links := FALSE;
		b_ausgefaedelt:=FALSE;
	END_IF
	IF 	b_materialmangel_rechts AND
		NOT fb_tof_bandende_re.Q   THEN
		b_materialmangel_rechts := FALSE;
		b_ausgefaedelt:=FALSE;
	END_IF
ELSE
	IF	gi16_maschinenstatusinfo = STATUS_MASCHINE_ARBEITET THEN
		IF 	NOT fb_tof_bandende_li.Q  AND zyl_bawe_querschub.fb.e_sensor1_eingefahren THEN
			b_materialmangel_links := TRUE;
		END_IF
		IF	NOT fb_tof_bandende_re.Q  AND zyl_bawe_querschub.fb.e_sensor1_ausgefahren THEN
			b_materialmangel_rechts := TRUE;
		END_IF
	END_IF
END_IF

(* ======================================Schrittkette======================================== *)
fb_state_entry(
	i16_next_step:= , 
	i16_pos:= 1,
	s_debugtext:= ,
	E=> ,
	X=> ,
	i16_step=> ,
	i16_last_step=> );

CASE fb_state_entry.i16_step OF
(*=======================================================*)
	INIT_OBJ:
		IF st_config.b_config_fertig THEN
			fb_state_entry.i16_next_step := INIT;
		END_IF

(*=======================================================*)
	INIT:
		IF fb_state_entry.E THEN
			fb_ton_wz.IN := FALSE;
			fb_ton_uez.IN	:= FALSE;
			fb_ton_quitt.IN := FALSE;
			sm_halter_nicht_oben := FALSE;
			sm_bandwechsel_ohne_ende := FALSE;
			sm_kein_band_anderer_einzug := FALSE;
			sm_kein_band_in_akt_einzug := FALSE;
			bm_bandwechselvorgang := FALSE;
			bm_bandwechsel_manuell := FALSE;
			st_ctrl_out.b_fehler := FALSE;
			st_ctrl_out.b_bereit := FALSE;
			st_ctrl_out.b_fertig := FALSE;
			st_ctrl_out.b_fertig_2 := FALSE;
			i16_vorgabe_ausfaedeln := 5;
			zyl_bawe_vorschub.st_ctrl.in.b_einfahren := FALSE;
			zyl_bawe_vorschub.st_ctrl.in.b_ausfahren := FALSE;
			zyl_bawe_querschub.st_ctrl.in.b_einfahren := FALSE;
			zyl_bawe_querschub.st_ctrl.in.b_ausfahren := FALSE;
			zyl_bawe_faenger_li.st_ctrl.in.b_einfahren := FALSE;
			zyl_bawe_faenger_li.st_ctrl.in.b_ausfahren := FALSE;
			zyl_bawe_faenger_re.st_ctrl.in.b_einfahren := FALSE;
			zyl_bawe_faenger_re.st_ctrl.in.b_ausfahren := FALSE;
			zyl_bawe_halter_li.st_ctrl.in.b_einfahren := FALSE;
			zyl_bawe_halter_li.st_ctrl.in.b_ausfahren := FALSE;
			zyl_bawe_halter_re.st_ctrl.in.b_einfahren := FALSE;
			zyl_bawe_halter_re.st_ctrl.in.b_ausfahren := FALSE;
			zyl_haspel_verschieben.st_ctrl.in.b_einfahren := FALSE;
			zyl_haspel_verschieben.st_ctrl.in.b_ausfahren := FALSE;
			zyl_bandeinzuege_verschieben.st_ctrl.in.b_einfahren := FALSE;
			zyl_bandeinzuege_verschieben.st_ctrl.in.b_ausfahren := FALSE;
			axis_bandeinzug_achse.st_ctrl.in.b_startpos := FALSE;
			visu_hinten.in.b_bandwechsel_aktiv := FALSE;
			b_materialmangel_links := FALSE;
			b_materialmangel_rechts := FALSE;
			b_ausgefaedelt:=FALSE;
			b_spulenwechsel:=FALSE;

			IF gst_datensatz.st_wkz.i16_typ_bandeinzug = SERVO THEN
				i16_vorgabe_einfaedeln :=2;
			ELSE
				i16_vorgabe_einfaedeln := gst_datensatz.st_wkz.i16_vorgabe_einfaedeln;
			END_IF
		END_IF

		(*-----------------------Weiterschaltbedingungen----------------------------*)
		IF st_ctrl_in.b_init THEN
			zyl_bawe_vorschub.st_ctrl.in.b_quittieren := FALSE;
			zyl_bawe_querschub.st_ctrl.in.b_quittieren := FALSE;
			zyl_bawe_faenger_li.st_ctrl.in.b_quittieren := FALSE;
			zyl_bawe_faenger_re.st_ctrl.in.b_quittieren := FALSE;
			zyl_bawe_halter_li.st_ctrl.in.b_quittieren := FALSE;
			zyl_bawe_halter_re.st_ctrl.in.b_quittieren := FALSE;
			zyl_haspel_verschieben.st_ctrl.in.b_quittieren := FALSE;
			zyl_bandeinzuege_verschieben.st_ctrl.in.b_quittieren := FALSE;

			IF NOT gst_datensatz.st_md.b_wt_transport_simulation THEN
				fb_state_entry.i16_next_step := 20;
			ELSE
				fb_state_entry.i16_next_step := BEREIT;
			END_IF
		END_IF

(*=======================================================*)
	20:	(* Abfrage Stellung Bandwechselquerschub  *)

		(*-----------------------Weiterschaltbedingungen----------------------------*)
		IF zyl_bawe_querschub.fb.e_sensor1_eingefahren THEN
			fb_state_entry.i16_next_step := 30;
		ELSIF zyl_bawe_querschub.fb.e_sensor1_ausgefahren THEN
			fb_state_entry.i16_next_step := 60;
		ELSE
			fb_state_entry.i16_next_step := 30;
		END_IF

(*=======================================================*)
	30:	(* Bandwechselquerschub einfahren *)
		IF fb_state_entry.E THEN
			zyl_bawe_querschub.st_ctrl.in.b_einfahren := TRUE;
		END_IF

		(*-----------------------Weiterschaltbedingungen----------------------------*)
		IF zyl_bawe_querschub.st_ctrl.out.b_eingefahren THEN
			zyl_bawe_querschub.st_ctrl.in.b_einfahren := FALSE;
			fb_state_entry.i16_next_step := 40;
		END_IF

(*=======================================================*)
	40:	(* Haspeln rechts: Haspel verschieben einfahren und Bandabzug ausfahren *)
		IF fb_state_entry.E THEN
			zyl_haspel_verschieben.st_ctrl.in.b_einfahren := TRUE;
			zyl_bandeinzuege_verschieben.st_ctrl.in.b_ausfahren := TRUE;
		END_IF
		(*-----------------------Weiterschaltbedingungen----------------------------*)
		IF  	zyl_haspel_verschieben.st_ctrl.out.b_eingefahren AND
 			zyl_bandeinzuege_verschieben.st_ctrl.out.b_ausgefahren
			THEN
				zyl_haspel_verschieben.st_ctrl.in.b_einfahren := FALSE;
				zyl_bandeinzuege_verschieben.st_ctrl.in.b_ausfahren := FALSE;
				fb_state_entry.i16_next_step := 50;
		END_IF

(*=======================================================*)
	50:	(* Halter rechts ausfahren und Band heben, Halter links einfahren  *)
		IF fb_state_entry.E THEN
			zyl_bawe_halter_re.st_ctrl.in.b_ausfahren := TRUE;
			zyl_bawe_halter_li.st_ctrl.in.b_einfahren := TRUE;
		END_IF

		(*-----------------------Weiterschaltbedingungen----------------------------*)
		IF 	zyl_bawe_halter_re.st_ctrl.out.b_ausgefahren AND
			zyl_bawe_halter_li.st_ctrl.out.b_eingefahren
			THEN
				zyl_bawe_halter_re.st_ctrl.in.b_ausfahren := FALSE;
				zyl_bawe_halter_li.st_ctrl.in.b_einfahren := FALSE;
				fb_state_entry.i16_next_step := 90;
		END_IF

(*=======================================================*)
	60:	(* Bandwechselquerschub ausfahren *)
		IF fb_state_entry.E THEN
			zyl_bawe_querschub.st_ctrl.in.b_ausfahren := TRUE;
		END_IF

		(*-----------------------Weiterschaltbedingungen----------------------------*)
		IF zyl_bawe_querschub.st_ctrl.out.b_ausgefahren THEN
			zyl_bawe_querschub.st_ctrl.in.b_ausfahren := FALSE;
			fb_state_entry.i16_next_step := 70;
		END_IF

(*=======================================================*)
	70:	(* Haspeln links: Haspel verschieben ausfahren und Bandabzug einfahren *)
		IF fb_state_entry.E THEN
			zyl_haspel_verschieben.st_ctrl.in.b_ausfahren := TRUE;
			zyl_bandeinzuege_verschieben.st_ctrl.in.b_einfahren := TRUE;
		END_IF
		(*-----------------------Weiterschaltbedingungen----------------------------*)
		IF  	zyl_haspel_verschieben.st_ctrl.out.b_ausgefahren AND
 			zyl_bandeinzuege_verschieben.st_ctrl.out.b_eingefahren
			THEN
				zyl_haspel_verschieben.st_ctrl.in.b_ausfahren := FALSE;
				zyl_bandeinzuege_verschieben.st_ctrl.in.b_einfahren := FALSE;
				fb_state_entry.i16_next_step := 80;
		END_IF

(*=======================================================*)
	80:	(* Halter links ausfahren und Band heben, Halter rechts einfahren  *)
		IF fb_state_entry.E THEN
			zyl_bawe_halter_li.st_ctrl.in.b_ausfahren := TRUE;
			zyl_bawe_halter_re.st_ctrl.in.b_einfahren := TRUE;
		END_IF

		(*-----------------------Weiterschaltbedingungen----------------------------*)
		IF 	zyl_bawe_halter_li.st_ctrl.out.b_ausgefahren AND
			zyl_bawe_halter_re.st_ctrl.out.b_eingefahren
			THEN
				zyl_bawe_halter_li.st_ctrl.in.b_ausfahren := FALSE;
				zyl_bawe_halter_re.st_ctrl.in.b_einfahren := FALSE;
				fb_state_entry.i16_next_step := 90;
		END_IF

(*=======================================================*)
	90:	(* Fänger links und rechts einfahren, damit Vorschub nach vorne fahren kann *)
		IF fb_state_entry.E THEN
			zyl_bawe_faenger_li.st_ctrl.in.b_einfahren := TRUE;
			zyl_bawe_faenger_re.st_ctrl.in.b_einfahren := TRUE;
		END_IF

		(*-----------------------Weiterschaltbedingungen----------------------------*)
		IF 	zyl_bawe_faenger_li.st_ctrl.out.b_eingefahren AND
			zyl_bawe_faenger_re.st_ctrl.out.b_eingefahren
			THEN
				zyl_bawe_faenger_li.st_ctrl.in.b_einfahren := FALSE;
				zyl_bawe_faenger_re.st_ctrl.in.b_einfahren := FALSE;
				fb_state_entry.i16_next_step := 95;
		END_IF

(*=======================================================*)
	95:	(* Vorschub ausfahren *)
		IF fb_state_entry.E THEN
			zyl_bawe_vorschub.st_ctrl.in.b_ausfahren := TRUE;
		END_IF

		(*-----------------------Weiterschaltbedingungen----------------------------*)
		IF zyl_bawe_vorschub.st_ctrl.out.b_ausgefahren THEN
			zyl_bawe_vorschub.st_ctrl.in.b_ausfahren := FALSE;
			fb_state_entry.i16_next_step := BEREIT;
		END_IF

(*=======================================================*)
	BEREIT:
		IF fb_state_entry.E THEN
			st_ctrl_out.b_bereit := TRUE;
			i16_akt_einfaedeln := 0;
			i16_akt_ausfaedeln := 0;
			bm_bandwechselvorgang := FALSE;
		END_IF

		(*-----------------------Weiterschaltbedingungen----------------------------*)
		(* Warte darauf, das ein Band leer wird und Starte Teil 1 zum Bandausfädeln *)
		(* Freigaben bei installietem Barcodereader wieder rein *)
		IF fb_r_trig_start.Q OR fb_r_trig_ibn_start.Q THEN
			st_ctrl_out.b_fertig := FALSE;
			st_ctrl_out.b_fertig_2 := FALSE;
			(* Nach dem Bandwechsel soll die Maschine in Einzelfertigung gehen*)
			IF NOT fb_tof_bandende_li.Q  AND zyl_bawe_querschub.fb.e_sensor1_eingefahren (*AND gst_barcode_persistent.b_band_rechts_ok*) THEN
				bm_bandwechselvorgang := TRUE;
				(* Nach dem Bandwechsel geht die Maschine in Abhängigkeit der Bedienereinstellung auf der Visu in Einzelfertigung *)
				fb_state_entry.i16_next_step := 200;
			ELSIF NOT fb_tof_bandende_re.Q  AND zyl_bawe_querschub.fb.e_sensor1_ausgefahren (* AND gst_barcode_persistent.b_band_links_ok*) THEN
				bm_bandwechselvorgang := TRUE;
				(* Nach dem Bandwechsel geht die Maschine in Abhängigkeit der Bedienereinstellung auf der Visu in Einzelfertigung *)
				fb_state_entry.i16_next_step := 500;
			ELSE
				sm_bandwechsel_ohne_ende := TRUE;
				fb_state_entry.i16_next_step := FEHLER;
			END_IF
		END_IF


(*---------------------------------------------------------------------------------------------------------------------------------------------------------------------------------------------------*)
(*========================Bandeinzug links ist leer===============================*)
	200:	(* Fänger links ausfahren zum Band halten, Fänger rechts einfahren zur Bandfreigabe im rechten Einzug - Halter gegensinnig *)
		IF fb_state_entry.E THEN
			zyl_bawe_faenger_li.st_ctrl.in.b_ausfahren := TRUE;
			zyl_bawe_faenger_re.st_ctrl.in.b_einfahren := TRUE;
			zyl_bawe_halter_li.st_ctrl.in.b_einfahren := TRUE;
			zyl_bawe_halter_re.st_ctrl.in.b_ausfahren := TRUE;
		END_IF

		(*-----------------------Weiterschaltbedingungen----------------------------*)
		IF 	zyl_bawe_faenger_li.st_ctrl.out.b_ausgefahren AND
			zyl_bawe_faenger_re.st_ctrl.out.b_eingefahren AND
			zyl_bawe_halter_li.st_ctrl.out.b_eingefahren AND
			zyl_bawe_halter_re.st_ctrl.out.b_ausgefahren AND
			gb_ba_auto_kontroller
			THEN
				zyl_bawe_faenger_li.st_ctrl.in.b_ausfahren := FALSE;
				zyl_bawe_faenger_re.st_ctrl.in.b_einfahren := FALSE;
				zyl_bawe_halter_li.st_ctrl.in.b_einfahren := FALSE;
				zyl_bawe_halter_re.st_ctrl.in.b_ausfahren := FALSE;
				fb_state_entry.i16_next_step := 210;
		END_IF

(*=======================================================*)
	210:	(* Band-Zylinder einfahren bzw. Servobandeinzug lösen *)
		CASE gst_datensatz.st_wkz.i16_typ_bandeinzug OF

			BANDWECHSLER_V2:
				IF fb_state_entry.E THEN
					(* Zylinder einfahren *)
					zyl_bandfaenger.st_ctrl.in.b_einfahren := TRUE;
					zyl_bandklemmen.st_ctrl.in.b_einfahren := TRUE;
				END_IF
					(* Bandwechsler V2 ohne Sensoren und anderen Zylindern *)
					gst_datensatz.st_wkz.nockenschaltwerk_bestueckachse.arr_nocken[NO_BW_BANDFAENGER_BAWEV2_EINFAHREN].b_camvalid := FALSE;
					gst_datensatz.st_wkz.nockenschaltwerk_bestueckachse.arr_nocken[NO_BW_BANDFAENGER_BAWEV2_AUSFAHREN].b_camvalid := FALSE;
					gst_datensatz.st_wkz.nockenschaltwerk_bestueckachse.arr_nocken[NO_BW_BANDKLEMMEN_BAWEV2_EINFAHREN].b_camvalid := FALSE;
					gst_datensatz.st_wkz.nockenschaltwerk_bestueckachse.arr_nocken[NO_BW_BANDKLEMMEN_BAWEV2_AUSFAHREN].b_camvalid := FALSE;
				(*-----------------------Weiterschaltbedingungen----------------------------*)
				IF 	zyl_bandfaenger.st_ctrl.out.b_eingefahren AND
					zyl_bandklemmen.st_ctrl.out.b_eingefahren AND
					gb_ba_auto_kontroller
					THEN
						zyl_bandfaenger.st_ctrl.in.b_einfahren := FALSE;
						zyl_bandklemmen.st_ctrl.in.b_einfahren := FALSE;
						fb_state_entry.i16_next_step := 220;
				END_IF

			SERVO:
				zyl_bawe_faenger_li.st_ctrl.in.b_einfahren := TRUE;
				zyl_bawe_halter_li.st_ctrl.in.b_einfahren := TRUE;
				(*-----------------------Weiterschaltbedingungen----------------------------*)
				IF 	zyl_bawe_faenger_li.st_ctrl.out.b_eingefahren AND
					zyl_bawe_halter_li.st_ctrl.out.b_eingefahren AND
					gb_ba_auto_kontroller
					THEN
						zyl_bawe_faenger_li.st_ctrl.in.b_einfahren := FALSE;
						zyl_bawe_halter_li.st_ctrl.in.b_einfahren := FALSE;
						fb_state_entry.i16_next_step := 216;
				END_IF
		END_CASE;

